LIN {X 0,Y 165.285,Z 372.711,A -85,B 0,C 180,E1 -23309.997,E2 -23309.997} C_VEL
LIN {X 0,Y 164.769,Z 372.772,A -85,B 0,C 180,E1 -23314.891,E2 -23314.891} C_VEL
LIN {X 0,Y 164.844,Z 372.763,A -85,B 0,C 180,E1 -23319.816,E2 -23319.816} C_VEL
LIN {X 0,Y 164.543,Z 372.8,A -85,B 0,C 180,E1 -23324.846,E2 -23324.846} C_VEL
LIN {X 0,Y 164.463,Z 372.807,A -85,B 0,C 180,E1 -23329.987,E2 -23329.987} C_VEL
LIN {X 0,Y 164.382,Z 372.819,A -85,B 0,C 180,E1 -23336.132,E2 -23336.132} C_VEL
LIN {X 0,Y 164.364,Z 372.823,A -85,B 0,C 180,E1 -23341.227,E2 -23341.227} C_VEL
LIN {X 0,Y 164.341,Z 372.821,A -85,B 0,C 180,E1 -23346.773,E2 -23346.773} C_VEL
LIN {X 0,Y 164.367,Z 372.822,A -85,B 0,C 180,E1 -23349.889,E2 -23349.889} C_VEL
LIN {X 0,Y 164.382,Z 372.818,A -85,B 0,C 180,E1 -23353.384,E2 -23353.384} C_VEL
LIN {X 0,Y 164.385,Z 372.819,A -85,B 0,C 180,E1 -23356.843,E2 -23356.843} C_VEL
LIN {X 0,Y 164.365,Z 372.822,A -85,B 0,C 180,E1 -23360.317,E2 -23360.317} C_VEL
LIN {X 0,Y 164.336,Z 372.823,A -85,B 0,C 180,E1 -23364.34,E2 -23364.34} C_VEL
LIN {X 0,Y 164.379,Z 372.819,A -85,B 0,C 180,E1 -23369.135,E2 -23369.135} C_VEL
LIN {X 0,Y 164.413,Z 372.819,A -85,B 0,C 180,E1 -23374.697,E2 -23374.697} C_VEL
LIN {X 0,Y 164.509,Z 372.8,A -85,B 0,C 180,E1 -23380.018,E2 -23380.018} C_VEL
LIN {X 0,Y 164.551,Z 372.798,A -85,B 0,C 180,E1 -23385.154,E2 -23385.154} C_VEL
LIN {X 0,Y 164.842,Z 372.763,A -85,B 0,C 180,E1 -23390.183,E2 -23390.183} C_VEL
LIN {X 0,Y 164.852,Z 372.762,A -85,B 0,C 180,E1 -23392.654,E2 -23392.654} C_VEL
LIN {X 0,Y 165.041,Z 372.736,A -85,B 0,C 180,E1 -23397.562,E2 -23397.562} C_VEL
LIN {X 0,Y 165.286,Z 372.71,A -85,B 0,C 180,E1 -23400.002,E2 -23400.002} C_VEL
LIN {X 0,Y 164.768,Z 372.768,A -85,B 0,C 180,E1 -23404.896,E2 -23404.896} C_VEL
LIN {X 0,Y 164.853,Z 372.762,A -85,B 0,C 180,E1 -23407.35,E2 -23407.35} C_VEL
LIN {X 0,Y 164.742,Z 372.774,A -85,B 0,C 180,E1 -23411.148,E2 -23411.148} C_VEL
LIN {X 0,Y 164.491,Z 372.809,A -85,B 0,C 180,E1 -23417.405,E2 -23417.405} C_VEL
LIN {X 0,Y 164.468,Z 372.806,A -85,B 0,C 180,E1 -23419.992,E2 -23419.992} C_VEL
LIN {X 0,Y 164.388,Z 372.819,A -85,B 0,C 180,E1 -23426.137,E2 -23426.137} C_VEL
LIN {X 0,Y 164.37,Z 372.822,A -85,B 0,C 180,E1 -23431.232,E2 -23431.232} C_VEL
LIN {X 0,Y 164.29,Z 372.83,A -85,B 0,C 180,E1 -23436.793,E2 -23436.793} C_VEL
LIN {X 0,Y 164.289,Z 372.831,A -85,B 0,C 180,E1 -23439.919,E2 -23439.919} C_VEL
LIN {X 0,Y 164.529,Z 372.877,A -85,B 0,C 180,E1 -23446.125,E2 -23446.125} C_VEL
LIN {X 0,Y 165.393,Z 377.162,A -85,B 0,C 180,E1 -23451.969,E2 -23451.969} C_VEL
LIN {X 0,Y 165.659,Z 379.629,A -85,B 0,C 180,E1 -23455.155,E2 -23455.155} C_VEL
LIN {X 0,Y 164.918,Z 382.338,A -85,B 0,C 180,E1 -23458.467,E2 -23458.467} C_VEL
LIN {X 0,Y 163.951,Z 385.365,A -85,B 0,C 180,E1 -23462.135,E2 -23462.135} C_VEL
LIN {X 0,Y 165.313,Z 398.175,A -85,B 0,C 180,E1 -23463.679,E2 -23463.679} C_VEL
LIN {X 0,Y 166.01,Z 408.279,A -85,B 0,C 180,E1 -23465.292,E2 -23465.292} C_VEL
LIN {X 0,Y 166.358,Z 416.947,A -85,B 0,C 180,E1 -23467.001,E2 -23467.001} C_VEL
LIN {X 0,Y 166.469,Z 426.075,A -85,B 0,C 180,E1 -23469.194,E2 -23469.194} C_VEL
LIN {X 0,Y 166.277,Z 432.989,A -85,B 0,C 180,E1 -23471.202,E2 -23471.202} C_VEL
LIN {X 0,Y 164.707,Z 440.811,A -85,B 0,C 180,E1 -23473.901,E2 -23473.901} C_VEL
LIN {X 0,Y 163.462,Z 447.658,A -85,B 0,C 180,E1 -23476.958,E2 -23476.958} C_VEL
LIN {X 0,Y 162.683,Z 453.124,A -85,B 0,C 180,E1 -23480.053,E2 -23480.053} C_VEL
LIN {X 0,Y 162.191,Z 458.179,A -85,B 0,C 180,E1 -23483.784,E2 -23483.784} C_VEL
LIN {X 0,Y 162.156,Z 461.833,A -85,B 0,C 180,E1 -23487.519,E2 -23487.519} C_VEL
LIN {X 0,Y 162.287,Z 463.452,A -85,B 0,C 180,E1 -23490.003,E2 -23490.003} C_VEL
LIN {X 0,Y 161.97,Z 464.904,A -85,B 0,C 180,E1 -23493.61,E2 -23493.61} C_VEL
LIN {X 0,Y 162.138,Z 465.306,A -85,B 0,C 180,E1 -23497.475,E2 -23497.475} C_VEL
LIN {X 0,Y 162.598,Z 464.896,A -85,B 0,C 180,E1 -23499.959,E2 -23499.959} C_VEL
LIN {X 0,Y 163.324,Z 464.018,A -85,B 0,C 180,E1 -23502.428,E2 -23502.428} C_VEL
LIN {X 0,Y 164.353,Z 462.7,A -85,B 0,C 180,E1 -23504.87,E2 -23504.87} C_VEL
LIN {X 0,Y 166.476,Z 459.738,A -85,B 0,C 180,E1 -23508.462,E2 -23508.462} C_VEL
LIN {X 0,Y 169.37,Z 455.573,A -85,B 0,C 180,E1 -23511.932,E2 -23511.932} C_VEL
LIN {X 0,Y 172.955,Z 450.071,A -85,B 0,C 180,E1 -23515.259,E2 -23515.259} C_VEL
LIN {X 0,Y 175.939,Z 444.205,A -85,B 0,C 180,E1 -23517.996,E2 -23517.996} C_VEL
LIN {X 0,Y 178.202,Z 437.103,A -85,B 0,C 180,E1 -23520.847,E2 -23520.847} C_VEL
LIN {X 0,Y 179.47,Z 430.444,A -85,B 0,C 180,E1 -23523.249,E2 -23523.249} C_VEL
LIN {X 0,Y 180.203,Z 422.802,A -85,B 0,C 180,E1 -23525.807,E2 -23525.807} C_VEL
LIN {X 0,Y 180.245,Z 421.902,A -85,B 0,C 180,E1 -23526.094,E2 -23526.094} C_VEL
LIN {X 0,Y 180.072,Z 419.304,A -85,B 0,C 180,E1 -23527.031,E2 -23527.031} C_VEL
LIN {X 0,Y 179.317,Z 417.046,A -85,B 0,C 180,E1 -23528.033,E2 -23528.033} C_VEL
LIN {X 0,Y 176.917,Z 413.276,A -85,B 0,C 180,E1 -23530.156,E2 -23530.156} C_VEL
LIN {X 0,Y 172.898,Z 407.932,A -85,B 0,C 180,E1 -23533.533,E2 -23533.533} C_VEL
LIN {X 0,Y 171.927,Z 405.803,A -85,B 0,C 180,E1 -23534.644,E2 -23534.644} C_VEL
LIN {X 0,Y 169.122,Z 398.872,A -85,B 0,C 180,E1 -23538.422,E2 -23538.422} C_VEL
LIN {X 0,Y 167.171,Z 395.11,A -85,B 0,C 180,E1 -23540.902,E2 -23540.902} C_VEL
LIN {X 0,Y 166.686,Z 393.384,A -85,B 0,C 180,E1 -23541.849,E2 -23541.849} C_VEL
LIN {X 0,Y 164.248,Z 389.736,A -85,B 0,C 180,E1 -23545.195,E2 -23545.195} C_VEL
LIN {X 0,Y 163.031,Z 386.548,A -85,B 0,C 180,E1 -23547.664,E2 -23547.664} C_VEL
LIN {X 0,Y 159.813,Z 382.313,A -85,B 0,C 180,E1 -23555.65,E2 -23555.65} C_VEL
LIN {X 0,Y 159.422,Z 380.964,A -85,B 0,C 180,E1 -23560.691,E2 -23560.691} C_VEL
LIN {X 0,Y 160.286,Z 381.531,A -85,B 0,C 180,E1 -23566.625,E2 -23566.625} C_VEL
LIN {X 0,Y 163.146,Z 383.354,A -85,B 0,C 180,E1 -23572.806,E2 -23572.806} C_VEL
LIN {X 0,Y 164.296,Z 385.761,A -85,B 0,C 180,E1 -23575.09,E2 -23575.09} C_VEL
LIN {X 0,Y 167.058,Z 388.467,A -85,B 0,C 180,E1 -23578.791,E2 -23578.791} C_VEL
LIN {X 0,Y 171.293,Z 396.943,A -85,B 0,C 180,E1 -23584.704,E2 -23584.704} C_VEL
LIN {X 0,Y 173.349,Z 401.847,A -85,B 0,C 180,E1 -23587.539,E2 -23587.539} C_VEL
LIN {X 0,Y 175.255,Z 408.041,A -85,B 0,C 180,E1 -23590.689,E2 -23590.689} C_VEL
LIN {X 0,Y 176.257,Z 414.922,A -85,B 0,C 180,E1 -23593.839,E2 -23593.839} C_VEL
LIN {X 0,Y 176.281,Z 421.806,A -85,B 0,C 180,E1 -23596.888,E2 -23596.888} C_VEL
LIN {X 0,Y 175.611,Z 426.875,A -85,B 0,C 180,E1 -23599.189,E2 -23599.189} C_VEL
LIN {X 0,Y 175.131,Z 428.204,A -85,B 0,C 180,E1 -23599.767,E2 -23599.767} C_VEL
LIN {X 0,Y 171.752,Z 433.94,A -85,B 0,C 180,E1 -23602.123,E2 -23602.123} C_VEL
LIN {X 0,Y 168.512,Z 438.818,A -85,B 0,C 180,E1 -23604.646,E2 -23604.646} C_VEL
LIN {X 0,Y 164.887,Z 443.625,A -85,B 0,C 180,E1 -23607.957,E2 -23607.957} C_VEL
LIN {X 0,Y 161.8,Z 447.187,A -85,B 0,C 180,E1 -23611.412,E2 -23611.412} C_VEL
LIN {X 0,Y 159.242,Z 449.625,A -85,B 0,C 180,E1 -23615.008,E2 -23615.008} C_VEL
LIN {X 0,Y 157.275,Z 450.962,A -85,B 0,C 180,E1 -23618.723,E2 -23618.723} C_VEL
LIN {X 0,Y 155.498,Z 451.005,A -85,B 0,C 180,E1 -23623.681,E2 -23623.681} C_VEL
LIN {X 0,Y 154.826,Z 450.049,A -85,B 0,C 180,E1 -23627.083,E2 -23627.083} C_VEL
LIN {X 0,Y 154.681,Z 447.051,A -85,B 0,C 180,E1 -23632.219,E2 -23632.219} C_VEL
LIN {X 0,Y 155.103,Z 443.465,A -85,B 0,C 180,E1 -23635.93,E2 -23635.93} C_VEL
LIN {X 0,Y 155.766,Z 439.558,A -85,B 0,C 180,E1 -23639.004,E2 -23639.004} C_VEL
LIN {X 0,Y 156.675,Z 434.938,A -85,B 0,C 180,E1 -23641.899,E2 -23641.899} C_VEL
LIN {X 0,Y 157.955,Z 428.745,A -85,B 0,C 180,E1 -23644.992,E2 -23644.992} C_VEL
LIN {X 0,Y 159.061,Z 423.19,A -85,B 0,C 180,E1 -23647.269,E2 -23647.269} C_VEL
LIN {X 0,Y 160.6,Z 415.517,A -85,B 0,C 180,E1 -23649.838,E2 -23649.838} C_VEL
LIN {X 0,Y 162.128,Z 407.481,A -85,B 0,C 180,E1 -23652.006,E2 -23652.006} C_VEL
LIN {X 0,Y 161.25,Z 398.757,A -85,B 0,C 180,E1 -23654.125,E2 -23654.125} C_VEL
LIN {X 0,Y 159.645,Z 387.621,A -85,B 0,C 180,E1 -23656.31,E2 -23656.31} C_VEL
LIN {X 0,Y 157.788,Z 377.801,A -85,B 0,C 180,E1 -23657.853,E2 -23657.853} C_VEL
LIN {X 0,Y 156.746,Z 373.773,A -85,B 0,C 180,E1 -23658.44,E2 -23658.44} C_VEL
LIN {X 0,Y 157.383,Z 373.696,A -85,B 0,C 180,E1 -23662.298,E2 -23662.298} C_VEL
LIN {X 0,Y 157.934,Z 373.626,A -85,B 0,C 180,E1 -23667.446,E2 -23667.446} C_VEL
LIN {X 0,Y 158.246,Z 373.588,A -85,B 0,C 180,E1 -23669.997,E2 -23669.997} C_VEL
LIN {X 0,Y 157.816,Z 373.64,A -85,B 0,C 180,E1 -23677.674,E2 -23677.674} C_VEL
LIN {X 0,Y 157.696,Z 373.65,A -85,B 0,C 180,E1 -23681.359,E2 -23681.359} C_VEL
LIN {X 0,Y 157.468,Z 373.683,A -85,B 0,C 180,E1 -23685.529,E2 -23685.529} C_VEL
LIN {X 0,Y 157.359,Z 373.691,A -85,B 0,C 180,E1 -23690.931,E2 -23690.931} C_VEL
LIN {X 0,Y 157.303,Z 373.7,A -85,B 0,C 180,E1 -23696.683,E2 -23696.683} C_VEL
LIN {X 0,Y 157.266,Z 373.707,A -85,B 0,C 180,E1 -23702.425,E2 -23702.425} C_VEL
LIN {X 0,Y 157.315,Z 373.696,A -85,B 0,C 180,E1 -23706.477,E2 -23706.477} C_VEL
LIN {X 0,Y 157.287,Z 373.703,A -85,B 0,C 180,E1 -23712.081,E2 -23712.081} C_VEL
LIN {X 0,Y 157.302,Z 373.7,A -85,B 0,C 180,E1 -23715.626,E2 -23715.626} C_VEL
LIN {X 0,Y 157.28,Z 373.703,A -85,B 0,C 180,E1 -23721.279,E2 -23721.279} C_VEL
LIN {X 0,Y 157.283,Z 373.702,A -85,B 0,C 180,E1 -23724.49,E2 -23724.49} C_VEL
LIN {X 0,Y 157.282,Z 373.705,A -85,B 0,C 180,E1 -23728.095,E2 -23728.095} C_VEL
LIN {X 0,Y 157.315,Z 373.7,A -85,B 0,C 180,E1 -23733.468,E2 -23733.468} C_VEL
LIN {X 0,Y 157.435,Z 373.68,A -85,B 0,C 180,E1 -23739.617,E2 -23739.617} C_VEL
LIN {X 0,Y 157.479,Z 373.681,A -85,B 0,C 180,E1 -23744.471,E2 -23744.471} C_VEL
LIN {X 0,Y 157.762,Z 373.643,A -85,B 0,C 180,E1 -23749.738,E2 -23749.738} C_VEL
LIN {X 0,Y 157.814,Z 373.64,A -85,B 0,C 180,E1 -23752.325,E2 -23752.325} C_VEL
LIN {X 0,Y 158.248,Z 373.587,A -85,B 0,C 180,E1 -23760.003,E2 -23760.003} C_VEL
LIN {X 0,Y 157.812,Z 373.64,A -85,B 0,C 180,E1 -23767.68,E2 -23767.68} C_VEL
LIN {X 0,Y 157.671,Z 373.656,A -85,B 0,C 180,E1 -23771.317,E2 -23771.317} C_VEL
LIN {X 0,Y 157.456,Z 373.684,A -85,B 0,C 180,E1 -23775.536,E2 -23775.536} C_VEL
LIN {X 0,Y 157.365,Z 373.69,A -85,B 0,C 180,E1 -23780.936,E2 -23780.936} C_VEL
LIN {X 0,Y 157.309,Z 373.701,A -85,B 0,C 180,E1 -23786.688,E2 -23786.688} C_VEL
LIN {X 0,Y 157.27,Z 373.706,A -85,B 0,C 180,E1 -23792.431,E2 -23792.431} C_VEL
LIN {X 0,Y 157.263,Z 373.705,A -85,B 0,C 180,E1 -23796.453,E2 -23796.453} C_VEL
LIN {X 0,Y 157.226,Z 373.712,A -85,B 0,C 180,E1 -23802.109,E2 -23802.109} C_VEL
LIN {X 0,Y 157.506,Z 373.679,A -85,B 0,C 180,E1 -23806.016,E2 -23806.016} C_VEL
LIN {X 0,Y 158.271,Z 377.582,A -85,B 0,C 180,E1 -23811.567,E2 -23811.567} C_VEL
LIN {X 0,Y 158.589,Z 379.982,A -85,B 0,C 180,E1 -23814.827,E2 -23814.827} C_VEL
LIN {X 0,Y 157.992,Z 382.259,A -85,B 0,C 180,E1 -23817.742,E2 -23817.742} C_VEL
LIN {X 0,Y 157.051,Z 385.056,A -85,B 0,C 180,E1 -23821.296,E2 -23821.296} C_VEL
LIN {X 0,Y 158.389,Z 398.191,A -85,B 0,C 180,E1 -23822.981,E2 -23822.981} C_VEL
LIN {X 0,Y 158.988,Z 407.24,A -85,B 0,C 180,E1 -23824.473,E2 -23824.473} C_VEL
LIN {X 0,Y 159.316,Z 416.09,A -85,B 0,C 180,E1 -23826.267,E2 -23826.267} C_VEL
LIN {X 0,Y 159.441,Z 423.58,A -85,B 0,C 180,E1 -23828.097,E2 -23828.097} C_VEL
LIN {X 0,Y 159.372,Z 431.315,A -85,B 0,C 180,E1 -23830.355,E2 -23830.355} C_VEL
LIN {X 0,Y 158.554,Z 436.045,A -85,B 0,C 180,E1 -23831.928,E2 -23831.928} C_VEL
LIN {X 0,Y 157.334,Z 442.433,A -85,B 0,C 180,E1 -23834.457,E2 -23834.457} C_VEL
LIN {X 0,Y 156.328,Z 447.731,A -85,B 0,C 180,E1 -23837.013,E2 -23837.013} C_VEL
LIN {X 0,Y 155.696,Z 452.163,A -85,B 0,C 180,E1 -23839.601,E2 -23839.601} C_VEL
LIN {X 0,Y 155.259,Z 455.836,A -85,B 0,C 180,E1 -23842.199,E2 -23842.199} C_VEL
LIN {X 0,Y 155.08,Z 459.541,A -85,B 0,C 180,E1 -23845.59,E2 -23845.59} C_VEL
LIN {X 0,Y 155.084,Z 461.11,A -85,B 0,C 180,E1 -23847.406,E2 -23847.406} C_VEL
LIN {X 0,Y 155.224,Z 462.836,A -85,B 0,C 180,E1 -23850.003,E2 -23850.003} C_VEL
LIN {X 0,Y 154.902,Z 464.291,A -85,B 0,C 180,E1 -23853.453,E2 -23853.453} C_VEL
LIN {X 0,Y 155.083,Z 464.946,A -85,B 0,C 180,E1 -23857.817,E2 -23857.817} C_VEL
LIN {X 0,Y 155.605,Z 464.613,A -85,B 0,C 180,E1 -23860.412,E2 -23860.412} C_VEL
LIN {X 0,Y 156.381,Z 463.847,A -85,B 0,C 180,E1 -23862.989,E2 -23862.989} C_VEL
LIN {X 0,Y 157.499,Z 462.645,A -85,B 0,C 180,E1 -23865.533,E2 -23865.533} C_VEL
LIN {X 0,Y 159.756,Z 459.824,A -85,B 0,C 180,E1 -23869.268,E2 -23869.268} C_VEL
LIN {X 0,Y 162.809,Z 455.818,A -85,B 0,C 180,E1 -23872.865,E2 -23872.865} C_VEL
LIN {X 0,Y 165.249,Z 452.405,A -85,B 0,C 180,E1 -23875.173,E2 -23875.173} C_VEL
LIN {X 0,Y 168.524,Z 447.242,A -85,B 0,C 180,E1 -23877.947,E2 -23877.947} C_VEL
LIN {X 0,Y 170.516,Z 442.77,A -85,B 0,C 180,E1 -23880.052,E2 -23880.052} C_VEL
LIN {X 0,Y 172.512,Z 436.516,A -85,B 0,C 180,E1 -23882.673,E2 -23882.673} C_VEL
LIN {X 0,Y 173.884,Z 429.558,A -85,B 0,C 180,E1 -23885.331,E2 -23885.331} C_VEL
LIN {X 0,Y 174.626,Z 422.22,A -85,B 0,C 180,E1 -23887.929,E2 -23887.929} C_VEL
LIN {X 0,Y 174.673,Z 415.952,A -85,B 0,C 180,E1 -23890.138,E2 -23890.138} C_VEL
LIN {X 0,Y 173.783,Z 411.346,A -85,B 0,C 180,E1 -23892.037,E2 -23892.037} C_VEL
LIN {X 0,Y 171.927,Z 405.803,A -85,B 0,C 180,E1 -23894.644,E2 -23894.644} C_VEL
LIN {X 0,Y 170.991,Z 403.904,A -85,B 0,C 180,E1 -23895.746,E2 -23895.746} C_VEL
LIN {X 0,Y 169.743,Z 402.527,A -85,B 0,C 180,E1 -23896.911,E2 -23896.911} C_VEL
LIN {X 0,Y 166.812,Z 400.799,A -85,B 0,C 180,E1 -23899.354,E2 -23899.354} C_VEL
LIN {X 0,Y 162.748,Z 398.577,A -85,B 0,C 180,E1 -23903.254,E2 -23903.254} C_VEL
LIN {X 0,Y 161.832,Z 397.323,A -85,B 0,C 180,E1 -23904.566,E2 -23904.566} C_VEL
LIN {X 0,Y 160.311,Z 392.937,A -85,B 0,C 180,E1 -23908.257,E2 -23908.257} C_VEL
LIN {X 0,Y 158.195,Z 390.036,A -85,B 0,C 180,E1 -23913.621,E2 -23913.621} C_VEL
LIN {X 0,Y 157.387,Z 387.899,A -85,B 0,C 180,E1 -23919.683,E2 -23919.683} C_VEL
LIN {X 0,Y 157.738,Z 387.938,A -85,B 0,C 180,E1 -23924.492,E2 -23924.492} C_VEL
LIN {X 0,Y 159.273,Z 389.077,A -85,B 0,C 180,E1 -23929.832,E2 -23929.832} C_VEL
LIN {X 0,Y 160.494,Z 389.995,A -85,B 0,C 180,E1 -23932.449,E2 -23932.449} C_VEL
LIN {X 0,Y 162.076,Z 392.91,A -85,B 0,C 180,E1 -23935.852,E2 -23935.852} C_VEL
LIN {X 0,Y 163.235,Z 394.058,A -85,B 0,C 180,E1 -23937.53,E2 -23937.53} C_VEL
LIN {X 0,Y 164.6,Z 396.861,A -85,B 0,C 180,E1 -23939.998,E2 -23939.998} C_VEL
LIN {X 0,Y 167.475,Z 403.476,A -85,B 0,C 180,E1 -23944.812,E2 -23944.812} C_VEL
LIN {X 0,Y 169.413,Z 409.495,A -85,B 0,C 180,E1 -23948.455,E2 -23948.455} C_VEL
LIN {X 0,Y 170.37,Z 414.917,A -85,B 0,C 180,E1 -23951.297,E2 -23951.297} C_VEL
LIN {X 0,Y 170.554,Z 420.996,A -85,B 0,C 180,E1 -23954.312,E2 -23954.312} C_VEL
LIN {X 0,Y 170.038,Z 426.114,A -85,B 0,C 180,E1 -23956.815,E2 -23956.815} C_VEL
LIN {X 0,Y 169.16,Z 429.719,A -85,B 0,C 180,E1 -23958.591,E2 -23958.591} C_VEL
LIN {X 0,Y 165.611,Z 435.223,A -85,B 0,C 180,E1 -23960.988,E2 -23960.988} C_VEL
LIN {X 0,Y 161.643,Z 440.657,A -85,B 0,C 180,E1 -23964.063,E2 -23964.063} C_VEL
LIN {X 0,Y 158.138,Z 444.855,A -85,B 0,C 180,E1 -23967.266,E2 -23967.266} C_VEL
LIN {X 0,Y 155.123,Z 447.974,A -85,B 0,C 180,E1 -23970.586,E2 -23970.586} C_VEL
LIN {X 0,Y 152.617,Z 450.094,A -85,B 0,C 180,E1 -23974.009,E2 -23974.009} C_VEL
LIN {X 0,Y 150.657,Z 451.288,A -85,B 0,C 180,E1 -23977.525,E2 -23977.525} C_VEL
LIN {X 0,Y 149.076,Z 451.591,A -85,B 0,C 180,E1 -23981.297,E2 -23981.297} C_VEL
LIN {X 0,Y 147.984,Z 450.79,A -85,B 0,C 180,E1 -23985.424,E2 -23985.424} C_VEL
LIN {X 0,Y 147.529,Z 448.816,A -85,B 0,C 180,E1 -23989.655,E2 -23989.655} C_VEL
LIN {X 0,Y 147.569,Z 447.478,A -85,B 0,C 180,E1 -23991.744,E2 -23991.744} C_VEL
LIN {X 0,Y 147.884,Z 444.385,A -85,B 0,C 180,E1 -23995.226,E2 -23995.226} C_VEL
LIN {X 0,Y 148.78,Z 439.15,A -85,B 0,C 180,E1 -23999.479,E2 -23999.479} C_VEL
LIN {X 0,Y 149.55,Z 435.318,A -85,B 0,C 180,E1 -24001.966,E2 -24001.966} C_VEL
LIN {X 0,Y 150.855,Z 429.126,A -85,B 0,C 180,E1 -24005.207,E2 -24005.207} C_VEL
LIN {X 0,Y 152.018,Z 423.532,A -85,B 0,C 180,E1 -24007.604,E2 -24007.604} C_VEL
LIN {X 0,Y 153.327,Z 417.122,A -85,B 0,C 180,E1 -24009.89,E2 -24009.89} C_VEL
LIN {X 0,Y 154.956,Z 408.973,A -85,B 0,C 180,E1 -24012.25,E2 -24012.25} C_VEL
LIN {X 0,Y 155.068,Z 406.477,A -85,B 0,C 180,E1 -24012.935,E2 -24012.935} C_VEL
LIN {X 0,Y 153.893,Z 396.06,A -85,B 0,C 180,E1 -24015.45,E2 -24015.45} C_VEL
LIN {X 0,Y 152.541,Z 387.141,A -85,B 0,C 180,E1 -24017.219,E2 -24017.219} C_VEL
LIN {X 0,Y 150.857,Z 378.629,A -85,B 0,C 180,E1 -24018.646,E2 -24018.646} C_VEL
LIN {X 0,Y 149.857,Z 374.63,A -85,B 0,C 180,E1 -24019.32,E2 -24019.32} C_VEL
LIN {X 0,Y 150.268,Z 374.581,A -85,B 0,C 180,E1 -24021.931,E2 -24021.931} C_VEL
LIN {X 0,Y 150.849,Z 374.509,A -85,B 0,C 180,E1 -24027.326,E2 -24027.326} C_VEL
LIN {X 0,Y 151.205,Z 374.465,A -85,B 0,C 180,E1 -24029.997,E2 -24029.997} C_VEL
LIN {X 0,Y 150.754,Z 374.519,A -85,B 0,C 180,E1 -24038.036,E2 -24038.036} C_VEL
LIN {X 0,Y 150.625,Z 374.53,A -85,B 0,C 180,E1 -24041.542,E2 -24041.542} C_VEL
LIN {X 0,Y 150.373,Z 374.566,A -85,B 0,C 180,E1 -24046.282,E2 -24046.282} C_VEL
LIN {X 0,Y 150.34,Z 374.565,A -85,B 0,C 180,E1 -24050.79,E2 -24050.79} C_VEL
LIN {X 0,Y 150.233,Z 374.58,A -85,B 0,C 180,E1 -24057.28,E2 -24057.28} C_VEL
LIN {X 0,Y 150.207,Z 374.586,A -85,B 0,C 180,E1 -24062.633,E2 -24062.633} C_VEL
LIN {X 0,Y 150.227,Z 374.581,A -85,B 0,C 180,E1 -24067.453,E2 -24067.453} C_VEL
LIN {X 0,Y 150.228,Z 374.584,A -85,B 0,C 180,E1 -24071.543,E2 -24071.543} C_VEL
LIN {X 0,Y 150.278,Z 374.575,A -85,B 0,C 180,E1 -24075.457,E2 -24075.457} C_VEL
LIN {X 0,Y 150.226,Z 374.585,A -85,B 0,C 180,E1 -24079.088,E2 -24079.088} C_VEL
LIN {X 0,Y 150.228,Z 374.58,A -85,B 0,C 180,E1 -24082.677,E2 -24082.677} C_VEL
LIN {X 0,Y 150.207,Z 374.586,A -85,B 0,C 180,E1 -24087.366,E2 -24087.366} C_VEL
LIN {X 0,Y 150.235,Z 374.581,A -85,B 0,C 180,E1 -24092.717,E2 -24092.717} C_VEL
LIN {X 0,Y 150.379,Z 374.559,A -85,B 0,C 180,E1 -24099.169,E2 -24099.169} C_VEL
LIN {X 0,Y 150.388,Z 374.564,A -85,B 0,C 180,E1 -24103.719,E2 -24103.719} C_VEL
LIN {X 0,Y 150.678,Z 374.525,A -85,B 0,C 180,E1 -24109.25,E2 -24109.25} C_VEL
LIN {X 0,Y 150.752,Z 374.52,A -85,B 0,C 180,E1 -24111.963,E2 -24111.963} C_VEL
LIN {X 0,Y 151.209,Z 374.464,A -85,B 0,C 180,E1 -24120.003,E2 -24120.003} C_VEL
LIN {X 0,Y 150.748,Z 374.52,A -85,B 0,C 180,E1 -24128.042,E2 -24128.042} C_VEL
LIN {X 0,Y 150.606,Z 374.534,A -85,B 0,C 180,E1 -24131.51,E2 -24131.51} C_VEL
LIN {X 0,Y 150.364,Z 374.567,A -85,B 0,C 180,E1 -24136.289,E2 -24136.289} C_VEL
LIN {X 0,Y 150.346,Z 374.564,A -85,B 0,C 180,E1 -24140.797,E2 -24140.797} C_VEL
LIN {X 0,Y 150.239,Z 374.581,A -85,B 0,C 180,E1 -24147.286,E2 -24147.286} C_VEL
LIN {X 0,Y 150.21,Z 374.586,A -85,B 0,C 180,E1 -24152.636,E2 -24152.636} C_VEL
LIN {X 0,Y 150.169,Z 374.587,A -85,B 0,C 180,E1 -24157.477,E2 -24157.477} C_VEL
LIN {X 0,Y 150.161,Z 374.592,A -85,B 0,C 180,E1 -24161.515,E2 -24161.515} C_VEL
LIN {X 0,Y 150.488,Z 374.661,A -85,B 0,C 180,E1 -24166.187,E2 -24166.187} C_VEL
LIN {X 0,Y 151.26,Z 378.692,A -85,B 0,C 180,E1 -24172.177,E2 -24172.177} C_VEL
LIN {X 0,Y 151.48,Z 380.375,A -85,B 0,C 180,E1 -24174.558,E2 -24174.558} C_VEL
LIN {X 0,Y 151.124,Z 382.059,A -85,B 0,C 180,E1 -24176.837,E2 -24176.837} C_VEL
LIN {X 0,Y 150.118,Z 384.782,A -85,B 0,C 180,E1 -24180.465,E2 -24180.465} C_VEL
LIN {X 0,Y 151.402,Z 397.721,A -85,B 0,C 180,E1 -24182.159,E2 -24182.159} C_VEL
LIN {X 0,Y 151.982,Z 406.007,A -85,B 0,C 180,E1 -24183.575,E2 -24183.575} C_VEL
LIN {X 0,Y 152.322,Z 415.052,A -85,B 0,C 180,E1 -24185.469,E2 -24185.469} C_VEL
LIN {X 0,Y 152.438,Z 423.314,A -85,B 0,C 180,E1 -24187.569,E2 -24187.569} C_VEL
LIN {X 0,Y 152.347,Z 430.539,A -85,B 0,C 180,E1 -24189.762,E2 -24189.762} C_VEL
LIN {X 0,Y 151.83,Z 434.523,A -85,B 0,C 180,E1 -24191.098,E2 -24191.098} C_VEL
LIN {X 0,Y 150.465,Z 441.089,A -85,B 0,C 180,E1 -24193.729,E2 -24193.729} C_VEL
LIN {X 0,Y 149.216,Z 447.73,A -85,B 0,C 180,E1 -24197.076,E2 -24197.076} C_VEL
LIN {X 0,Y 148.449,Z 453.044,A -85,B 0,C 180,E1 -24200.466,E2 -24200.466} C_VEL
LIN {X 0,Y 148.079,Z 456.458,A -85,B 0,C 180,E1 -24203.189,E2 -24203.189} C_VEL
LIN {X 0,Y 148.027,Z 458.989,A -85,B 0,C 180,E1 -24205.612,E2 -24205.612} C_VEL
LIN {X 0,Y 148.16,Z 462.213,A -85,B 0,C 180,E1 -24210.003,E2 -24210.003} C_VEL
LIN {X 0,Y 147.844,Z 463.697,A -85,B 0,C 180,E1 -24213.341,E2 -24213.341} C_VEL
LIN {X 0,Y 147.843,Z 464.321,A -85,B 0,C 180,E1 -24215.459,E2 -24215.459} C_VEL
LIN {X 0,Y 148.037,Z 464.549,A -85,B 0,C 180,E1 -24218.192,E2 -24218.192} C_VEL
LIN {X 0,Y 148.608,Z 464.331,A -85,B 0,C 180,E1 -24220.908,E2 -24220.908} C_VEL
LIN {X 0,Y 149.465,Z 463.69,A -85,B 0,C 180,E1 -24223.601,E2 -24223.601} C_VEL
LIN {X 0,Y 150.652,Z 462.6,A -85,B 0,C 180,E1 -24226.258,E2 -24226.258} C_VEL
LIN {X 0,Y 153.075,Z 459.93,A -85,B 0,C 180,E1 -24230.145,E2 -24230.145} C_VEL
LIN {X 0,Y 156.3,Z 456.061,A -85,B 0,C 180,E1 -24233.875,E2 -24233.875} C_VEL
LIN {X 0,Y 160.27,Z 450.887,A -85,B 0,C 180,E1 -24237.419,E2 -24237.419} C_VEL
LIN {X 0,Y 162.821,Z 446.85,A -85,B 0,C 180,E1 -24239.624,E2 -24239.624} C_VEL
LIN {X 0,Y 165.124,Z 441.709,A -85,B 0,C 180,E1 -24242.144,E2 -24242.144} C_VEL
LIN {X 0,Y 166.951,Z 436.041,A -85,B 0,C 180,E1 -24244.635,E2 -24244.635} C_VEL
LIN {X 0,Y 168.436,Z 428.775,A -85,B 0,C 180,E1 -24247.552,E2 -24247.552} C_VEL
LIN {X 0,Y 169.213,Z 422.018,A -85,B 0,C 180,E1 -24250.142,E2 -24250.142} C_VEL
LIN {X 0,Y 169.101,Z 417.161,A -85,B 0,C 180,E1 -24252.149,E2 -24252.149} C_VEL
LIN {X 0,Y 167.294,Z 410.422,A -85,B 0,C 180,E1 -24255.579,E2 -24255.579} C_VEL
LIN {X 0,Y 164.999,Z 404.173,A -85,B 0,C 180,E1 -24259.271,E2 -24259.271} C_VEL
LIN {X 0,Y 163.008,Z 399.017,A -85,B 0,C 180,E1 -24262.869,E2 -24262.869} C_VEL
LIN {X 0,Y 161.832,Z 397.323,A -85,B 0,C 180,E1 -24264.566,E2 -24264.566} C_VEL
LIN {X 0,Y 160.543,Z 395.876,A -85,B 0,C 180,E1 -24266.545,E2 -24266.545} C_VEL
LIN {X 0,Y 158.987,Z 395.532,A -85,B 0,C 180,E1 -24268.6,E2 -24268.6} C_VEL
LIN {X 0,Y 155.455,Z 396.122,A -85,B 0,C 180,E1 -24274.329,E2 -24274.329} C_VEL
LIN {X 0,Y 155.077,Z 395.767,A -85,B 0,C 180,E1 -24275.803,E2 -24275.803} C_VEL
LIN {X 0,Y 154.837,Z 394.827,A -85,B 0,C 180,E1 -24278.706,E2 -24278.706} C_VEL
LIN {X 0,Y 154.892,Z 394.404,A -85,B 0,C 180,E1 -24282.344,E2 -24282.344} C_VEL
LIN {X 0,Y 155.624,Z 394.948,A -85,B 0,C 180,E1 -24286.948,E2 -24286.948} C_VEL
LIN {X 0,Y 156.81,Z 395.842,A -85,B 0,C 180,E1 -24290.421,E2 -24290.421} C_VEL
LIN {X 0,Y 157.539,Z 396.61,A -85,B 0,C 180,E1 -24292.306,E2 -24292.306} C_VEL
LIN {X 0,Y 158.417,Z 398.721,A -85,B 0,C 180,E1 -24294.907,E2 -24294.907} C_VEL
LIN {X 0,Y 159.844,Z 400.412,A -85,B 0,C 180,E1 -24297.478,E2 -24297.478} C_VEL
LIN {X 0,Y 161.535,Z 404.863,A -85,B 0,C 180,E1 -24301.318,E2 -24301.318} C_VEL
LIN {X 0,Y 163.268,Z 409.677,A -85,B 0,C 180,E1 -24304.936,E2 -24304.936} C_VEL
LIN {X 0,Y 164.523,Z 415.377,A -85,B 0,C 180,E1 -24308.596,E2 -24308.596} C_VEL
LIN {X 0,Y 164.85,Z 420.122,A -85,B 0,C 180,E1 -24311.304,E2 -24311.304} C_VEL
LIN {X 0,Y 164.519,Z 425.494,A -85,B 0,C 180,E1 -24314.216,E2 -24314.216} C_VEL
LIN {X 0,Y 163.489,Z 430.396,A -85,B 0,C 180,E1 -24316.865,E2 -24316.865} C_VEL
LIN {X 0,Y 162.433,Z 432.501,A -85,B 0,C 180,E1 -24317.839,E2 -24317.839} C_VEL
LIN {X 0,Y 158.002,Z 438.654,A -85,B 0,C 180,E1 -24320.911,E2 -24320.911} C_VEL
LIN {X 0,Y 153.76,Z 443.57,A -85,B 0,C 180,E1 -24324.288,E2 -24324.288} C_VEL
LIN {X 0,Y 150.015,Z 447.322,A -85,B 0,C 180,E1 -24327.933,E2 -24327.933} C_VEL
LIN {X 0,Y 147.49,Z 449.466,A -85,B 0,C 180,E1 -24330.933,E2 -24330.933} C_VEL
LIN {X 0,Y 144.344,Z 451.469,A -85,B 0,C 180,E1 -24335.748,E2 -24335.748} C_VEL
LIN {X 0,Y 142.443,Z 451.96,A -85,B 0,C 180,E1 -24339.893,E2 -24339.893} C_VEL
LIN {X 0,Y 141.133,Z 451.306,A -85,B 0,C 180,E1 -24344.195,E2 -24344.195} C_VEL
LIN {X 0,Y 140.441,Z 448.97,A -85,B 0,C 180,E1 -24349.412,E2 -24349.412} C_VEL
LIN {X 0,Y 140.558,Z 446.312,A -85,B 0,C 180,E1 -24353.125,E2 -24353.125} C_VEL
LIN {X 0,Y 141.017,Z 442.783,A -85,B 0,C 180,E1 -24356.751,E2 -24356.751} C_VEL
LIN {X 0,Y 141.872,Z 438.302,A -85,B 0,C 180,E1 -24360.301,E2 -24360.301} C_VEL
LIN {X 0,Y 143.37,Z 431.237,A -85,B 0,C 180,E1 -24364.597,E2 -24364.597} C_VEL
LIN {X 0,Y 145.025,Z 423.68,A -85,B 0,C 180,E1 -24368.049,E2 -24368.049} C_VEL
LIN {X 0,Y 146.313,Z 417.512,A -85,B 0,C 180,E1 -24370.349,E2 -24370.349} C_VEL
LIN {X 0,Y 148.053,Z 409.218,A -85,B 0,C 180,E1 -24372.855,E2 -24372.855} C_VEL
LIN {X 0,Y 147.82,Z 404.136,A -85,B 0,C 180,E1 -24374.282,E2 -24374.282} C_VEL
LIN {X 0,Y 146.719,Z 394.89,A -85,B 0,C 180,E1 -24376.528,E2 -24376.528} C_VEL
LIN {X 0,Y 145.448,Z 386.406,A -85,B 0,C 180,E1 -24378.243,E2 -24378.243} C_VEL
LIN {X 0,Y 143.749,Z 378.858,A -85,B 0,C 180,E1 -24379.582,E2 -24379.582} C_VEL
LIN {X 0,Y 142.942,Z 375.493,A -85,B 0,C 180,E1 -24380.196,E2 -24380.196} C_VEL
LIN {X 0,Y 143.415,Z 375.437,A -85,B 0,C 180,E1 -24384.372,E2 -24384.372} C_VEL
LIN {X 0,Y 144.162,Z 375.343,A -85,B 0,C 180,E1 -24389.996,E2 -24389.996} C_VEL
LIN {X 0,Y 143.676,Z 375.4,A -85,B 0,C 180,E1 -24398.435,E2 -24398.435} C_VEL
LIN {X 0,Y 143.562,Z 375.41,A -85,B 0,C 180,E1 -24401.755,E2 -24401.755} C_VEL
LIN {X 0,Y 143.306,Z 375.446,A -85,B 0,C 180,E1 -24407.109,E2 -24407.109} C_VEL
LIN {X 0,Y 143.266,Z 375.447,A -85,B 0,C 180,E1 -24411.252,E2 -24411.252} C_VEL
LIN {X 0,Y 143.179,Z 375.456,A -85,B 0,C 180,E1 -24417.935,E2 -24417.935} C_VEL
LIN {X 0,Y 143.159,Z 375.465,A -85,B 0,C 180,E1 -24423.435,E2 -24423.435} C_VEL
LIN {X 0,Y 143.121,Z 375.469,A -85,B 0,C 180,E1 -24429.665,E2 -24429.665} C_VEL
LIN {X 0,Y 143.172,Z 375.459,A -85,B 0,C 180,E1 -24433.406,E2 -24433.406} C_VEL
LIN {X 0,Y 143.159,Z 375.465,A -85,B 0,C 180,E1 -24437.418,E2 -24437.418} C_VEL
LIN {X 0,Y 143.157,Z 375.461,A -85,B 0,C 180,E1 -24441.759,E2 -24441.759} C_VEL
LIN {X 0,Y 143.174,Z 375.463,A -85,B 0,C 180,E1 -24447.323,E2 -24447.323} C_VEL
LIN {X 0,Y 143.154,Z 375.464,A -85,B 0,C 180,E1 -24453.782,E2 -24453.782} C_VEL
LIN {X 0,Y 143.333,Z 375.437,A -85,B 0,C 180,E1 -24459.929,E2 -24459.929} C_VEL
LIN {X 0,Y 143.377,Z 375.437,A -85,B 0,C 180,E1 -24465.816,E2 -24465.816} C_VEL
LIN {X 0,Y 143.592,Z 375.408,A -85,B 0,C 180,E1 -24468.713,E2 -24468.713} C_VEL
LIN {X 0,Y 143.674,Z 375.4,A -85,B 0,C 180,E1 -24471.564,E2 -24471.564} C_VEL
LIN {X 0,Y 144.168,Z 375.341,A -85,B 0,C 180,E1 -24480.003,E2 -24480.003} C_VEL
LIN {X 0,Y 143.667,Z 375.401,A -85,B 0,C 180,E1 -24488.442,E2 -24488.442} C_VEL
LIN {X 0,Y 143.54,Z 375.413,A -85,B 0,C 180,E1 -24491.716,E2 -24491.716} C_VEL
LIN {X 0,Y 143.302,Z 375.447,A -85,B 0,C 180,E1 -24497.116,E2 -24497.116} C_VEL
LIN {X 0,Y 143.271,Z 375.446,A -85,B 0,C 180,E1 -24501.259,E2 -24501.259} C_VEL
LIN {X 0,Y 143.185,Z 375.457,A -85,B 0,C 180,E1 -24507.941,E2 -24507.941} C_VEL
LIN {X 0,Y 143.16,Z 375.465,A -85,B 0,C 180,E1 -24513.437,E2 -24513.437} C_VEL
LIN {X 0,Y 143.063,Z 375.475,A -85,B 0,C 180,E1 -24519.693,E2 -24519.693} C_VEL
LIN {X 0,Y 143.436,Z 375.498,A -85,B 0,C 180,E1 -24526.184,E2 -24526.184} C_VEL
LIN {X 0,Y 144.056,Z 378.782,A -85,B 0,C 180,E1 -24531.317,E2 -24531.317} C_VEL
LIN {X 0,Y 144.374,Z 380.752,A -85,B 0,C 180,E1 -24534.262,E2 -24534.262} C_VEL
LIN {X 0,Y 144.253,Z 381.905,A -85,B 0,C 180,E1 -24535.922,E2 -24535.922} C_VEL
LIN {X 0,Y 143.228,Z 384.46,A -85,B 0,C 180,E1 -24539.504,E2 -24539.504} C_VEL
LIN {X 0,Y 144.42,Z 396.684,A -85,B 0,C 180,E1 -24541.161,E2 -24541.161} C_VEL
LIN {X 0,Y 145.058,Z 405.901,A -85,B 0,C 180,E1 -24542.824,E2 -24542.824} C_VEL
LIN {X 0,Y 145.361,Z 415.59,A -85,B 0,C 180,E1 -24544.982,E2 -24544.982} C_VEL
LIN {X 0,Y 145.414,Z 423.959,A -85,B 0,C 180,E1 -24547.258,E2 -24547.258} C_VEL
LIN {X 0,Y 145.272,Z 431.84,A -85,B 0,C 180,E1 -24549.841,E2 -24549.841} C_VEL
LIN {X 0,Y 143.641,Z 439.698,A -85,B 0,C 180,E1 -24552.932,E2 -24552.932} C_VEL
LIN {X 0,Y 142.281,Z 446.559,A -85,B 0,C 180,E1 -24556.434,E2 -24556.434} C_VEL
LIN {X 0,Y 141.451,Z 452.028,A -85,B 0,C 180,E1 -24559.989,E2 -24559.989} C_VEL
LIN {X 0,Y 140.935,Z 457.078,A -85,B 0,C 180,E1 -24564.28,E2 -24564.28} C_VEL
LIN {X 0,Y 140.937,Z 459.619,A -85,B 0,C 180,E1 -24567.145,E2 -24567.145} C_VEL
LIN {X 0,Y 141.096,Z 461.586,A -85,B 0,C 180,E1 -24570.004,E2 -24570.004} C_VEL
LIN {X 0,Y 140.779,Z 463.076,A -85,B 0,C 180,E1 -24573.156,E2 -24573.156} C_VEL
LIN {X 0,Y 140.78,Z 463.819,A -85,B 0,C 180,E1 -24575.734,E2 -24575.734} C_VEL
LIN {X 0,Y 141.012,Z 464.147,A -85,B 0,C 180,E1 -24578.603,E2 -24578.603} C_VEL
LIN {X 0,Y 141.636,Z 464.054,A -85,B 0,C 180,E1 -24581.452,E2 -24581.452} C_VEL
LIN {X 0,Y 142.557,Z 463.537,A -85,B 0,C 180,E1 -24584.274,E2 -24584.274} C_VEL
LIN {X 0,Y 143.839,Z 462.479,A -85,B 0,C 180,E1 -24587.051,E2 -24587.051} C_VEL
LIN {X 0,Y 146.41,Z 460.021,A -85,B 0,C 180,E1 -24591.105,E2 -24591.105} C_VEL
LIN {X 0,Y 149.845,Z 456.34,A -85,B 0,C 180,E1 -24594.972,E2 -24594.972} C_VEL
LIN {X 0,Y 152.57,Z 453.242,A -85,B 0,C 180,E1 -24597.432,E2 -24597.432} C_VEL
LIN {X 0,Y 156.182,Z 448.411,A -85,B 0,C 180,E1 -24600.417,E2 -24600.417} C_VEL
LIN {X 0,Y 159.126,Z 442.561,A -85,B 0,C 180,E1 -24603.512,E2 -24603.512} C_VEL
LIN {X 0,Y 161.111,Z 437.152,A -85,B 0,C 180,E1 -24606.082,E2 -24606.082} C_VEL
LIN {X 0,Y 163.085,Z 428.986,A -85,B 0,C 180,E1 -24609.604,E2 -24609.604} C_VEL
LIN {X 0,Y 163.818,Z 423.238,A -85,B 0,C 180,E1 -24612.034,E2 -24612.034} C_VEL
LIN {X 0,Y 163.59,Z 420.324,A -85,B 0,C 180,E1 -24613.427,E2 -24613.427} C_VEL
LIN {X 0,Y 162.209,Z 414.194,A -85,B 0,C 180,E1 -24616.966,E2 -24616.966} C_VEL
LIN {X 0,Y 160.613,Z 409.085,A -85,B 0,C 180,E1 -24620.383,E2 -24620.383} C_VEL
LIN {X 0,Y 159.276,Z 404.852,A -85,B 0,C 180,E1 -24623.434,E2 -24623.434} C_VEL
LIN {X 0,Y 157.921,Z 402.181,A -85,B 0,C 180,E1 -24626.176,E2 -24626.176} C_VEL
LIN {X 0,Y 157.431,Z 400.067,A -85,B 0,C 180,E1 -24628.021,E2 -24628.021} C_VEL
LIN {X 0,Y 156.529,Z 398.372,A -85,B 0,C 180,E1 -24630.401,E2 -24630.401} C_VEL
LIN {X 0,Y 155.077,Z 395.767,A -85,B 0,C 180,E1 -24635.803,E2 -24635.803} C_VEL
LIN {X 0,Y 154.621,Z 395.661,A -85,B 0,C 180,E1 -24637.976,E2 -24637.976} C_VEL
LIN {X 0,Y 153.941,Z 396.672,A -85,B 0,C 180,E1 -24640.137,E2 -24640.137} C_VEL
LIN {X 0,Y 152.462,Z 400.877,A -85,B 0,C 180,E1 -24645.928,E2 -24645.928} C_VEL
LIN {X 0,Y 152.639,Z 401.441,A -85,B 0,C 180,E1 -24647.422,E2 -24647.422} C_VEL
LIN {X 0,Y 153.256,Z 401.886,A -85,B 0,C 180,E1 -24649.428,E2 -24649.428} C_VEL
LIN {X 0,Y 154.154,Z 402.96,A -85,B 0,C 180,E1 -24652.136,E2 -24652.136} C_VEL
LIN {X 0,Y 156.067,Z 406.563,A -85,B 0,C 180,E1 -24657.416,E2 -24657.416} C_VEL
LIN {X 0,Y 157.516,Z 411.51,A -85,B 0,C 180,E1 -24661.865,E2 -24661.865} C_VEL
LIN {X 0,Y 158.573,Z 415.549,A -85,B 0,C 180,E1 -24665.083,E2 -24665.083} C_VEL
LIN {X 0,Y 159.231,Z 421.072,A -85,B 0,C 180,E1 -24668.884,E2 -24668.884} C_VEL
LIN {X 0,Y 158.969,Z 425.721,A -85,B 0,C 180,E1 -24671.728,E2 -24671.728} C_VEL
LIN {X 0,Y 158.265,Z 429.8,A -85,B 0,C 180,E1 -24674.133,E2 -24674.133} C_VEL
LIN {X 0,Y 157.586,Z 432.109,A -85,B 0,C 180,E1 -24675.518,E2 -24675.518} C_VEL
LIN {X 0,Y 156.551,Z 434.074,A -85,B 0,C 180,E1 -24676.511,E2 -24676.511} C_VEL
LIN {X 0,Y 151.763,Z 439.998,A -85,B 0,C 180,E1 -24679.756,E2 -24679.756} C_VEL
LIN {X 0,Y 148.491,Z 443.558,A -85,B 0,C 180,E1 -24682.246,E2 -24682.246} C_VEL
LIN {X 0,Y 144.4,Z 447.407,A -85,B 0,C 180,E1 -24685.975,E2 -24685.975} C_VEL
LIN {X 0,Y 140.889,Z 450.109,A -85,B 0,C 180,E1 -24689.919,E2 -24689.919} C_VEL
LIN {X 0,Y 138.053,Z 451.725,A -85,B 0,C 180,E1 -24694.051,E2 -24694.051} C_VEL
LIN {X 0,Y 135.618,Z 452.319,A -85,B 0,C 180,E1 -24698.978,E2 -24698.978} C_VEL
LIN {X 0,Y 134.33,Z 451.775,A -85,B 0,C 180,E1 -24702.902,E2 -24702.902} C_VEL
LIN {X 0,Y 133.478,Z 450.053,A -85,B 0,C 180,E1 -24707.483,E2 -24707.483} C_VEL
LIN {X 0,Y 133.382,Z 447.043,A -85,B 0,C 180,E1 -24712.214,E2 -24712.214} C_VEL
LIN {X 0,Y 133.774,Z 443.704,A -85,B 0,C 180,E1 -24715.963,E2 -24715.963} C_VEL
LIN {X 0,Y 134.736,Z 438.605,A -85,B 0,C 180,E1 -24720.293,E2 -24720.293} C_VEL
LIN {X 0,Y 136.289,Z 431.504,A -85,B 0,C 180,E1 -24724.818,E2 -24724.818} C_VEL
LIN {X 0,Y 137.996,Z 423.967,A -85,B 0,C 180,E1 -24728.433,E2 -24728.433} C_VEL
LIN {X 0,Y 139.552,Z 416.782,A -85,B 0,C 180,E1 -24731.2,E2 -24731.2} C_VEL
LIN {X 0,Y 141.064,Z 409.937,A -85,B 0,C 180,E1 -24733.349,E2 -24733.349} C_VEL
LIN {X 0,Y 140.88,Z 405.039,A -85,B 0,C 180,E1 -24734.813,E2 -24734.813} C_VEL
LIN {X 0,Y 139.868,Z 396.049,A -85,B 0,C 180,E1 -24737.131,E2 -24737.131} C_VEL
LIN {X 0,Y 138.542,Z 386.997,A -85,B 0,C 180,E1 -24739.086,E2 -24739.086} C_VEL
LIN {X 0,Y 136.559,Z 378.646,A -85,B 0,C 180,E1 -24740.673,E2 -24740.673} C_VEL
LIN {X 0,Y 136.018,Z 376.356,A -85,B 0,C 180,E1 -24741.079,E2 -24741.079} C_VEL
LIN {X 0,Y 136.673,Z 376.275,A -85,B 0,C 180,E1 -24747.049,E2 -24747.049} C_VEL
LIN {X 0,Y 137.116,Z 376.22,A -85,B 0,C 180,E1 -24749.996,E2 -24749.996} C_VEL
LIN {X 0,Y 136.6,Z 376.281,A -85,B 0,C 180,E1 -24758.875,E2 -24758.875} C_VEL
LIN {X 0,Y 136.483,Z 376.291,A -85,B 0,C 180,E1 -24761.954,E2 -24761.954} C_VEL
LIN {X 0,Y 136.242,Z 376.324,A -85,B 0,C 180,E1 -24768.025,E2 -24768.025} C_VEL
LIN {X 0,Y 136.187,Z 376.331,A -85,B 0,C 180,E1 -24771.746,E2 -24771.746} C_VEL
LIN {X 0,Y 136.089,Z 376.339,A -85,B 0,C 180,E1 -24778.614,E2 -24778.614} C_VEL
LIN {X 0,Y 136.072,Z 376.346,A -85,B 0,C 180,E1 -24784.616,E2 -24784.616} C_VEL
LIN {X 0,Y 136.095,Z 376.345,A -85,B 0,C 180,E1 -24789.236,E2 -24789.236} C_VEL
LIN {X 0,Y 136.107,Z 376.338,A -85,B 0,C 180,E1 -24793.71,E2 -24793.71} C_VEL
LIN {X 0,Y 136.106,Z 376.343,A -85,B 0,C 180,E1 -24797.839,E2 -24797.839} C_VEL
LIN {X 0,Y 136.108,Z 376.339,A -85,B 0,C 180,E1 -24801.715,E2 -24801.715} C_VEL
LIN {X 0,Y 136.081,Z 376.345,A -85,B 0,C 180,E1 -24805.716,E2 -24805.716} C_VEL
LIN {X 0,Y 136.137,Z 376.335,A -85,B 0,C 180,E1 -24812.318,E2 -24812.318} C_VEL
LIN {X 0,Y 136.267,Z 376.317,A -85,B 0,C 180,E1 -24818.84,E2 -24818.84} C_VEL
LIN {X 0,Y 136.284,Z 376.32,A -85,B 0,C 180,E1 -24825.061,E2 -24825.061} C_VEL
LIN {X 0,Y 136.491,Z 376.29,A -85,B 0,C 180,E1 -24828.117,E2 -24828.117} C_VEL
LIN {X 0,Y 136.598,Z 376.281,A -85,B 0,C 180,E1 -24831.124,E2 -24831.124} C_VEL
LIN {X 0,Y 137.125,Z 376.218,A -85,B 0,C 180,E1 -24840.003,E2 -24840.003} C_VEL
LIN {X 0,Y 136.591,Z 376.282,A -85,B 0,C 180,E1 -24848.882,E2 -24848.882} C_VEL
LIN {X 0,Y 136.483,Z 376.29,A -85,B 0,C 180,E1 -24851.958,E2 -24851.958} C_VEL
LIN {X 0,Y 136.24,Z 376.325,A -85,B 0,C 180,E1 -24858.033,E2 -24858.033} C_VEL
LIN {X 0,Y 136.193,Z 376.329,A -85,B 0,C 180,E1 -24861.754,E2 -24861.754} C_VEL
LIN {X 0,Y 136.095,Z 376.34,A -85,B 0,C 180,E1 -24868.621,E2 -24868.621} C_VEL
LIN {X 0,Y 136.066,Z 376.348,A -85,B 0,C 180,E1 -24874.625,E2 -24874.625} C_VEL
LIN {X 0,Y 136.032,Z 376.351,A -85,B 0,C 180,E1 -24879.205,E2 -24879.205} C_VEL
LIN {X 0,Y 136.365,Z 376.326,A -85,B 0,C 180,E1 -24886.185,E2 -24886.185} C_VEL
LIN {X 0,Y 137.045,Z 379.901,A -85,B 0,C 180,E1 -24892.025,E2 -24892.025} C_VEL
LIN {X 0,Y 137.169,Z 382.276,A -85,B 0,C 180,E1 -24895.7,E2 -24895.7} C_VEL
LIN {X 0,Y 136.394,Z 384.173,A -85,B 0,C 180,E1 -24898.503,E2 -24898.503} C_VEL
LIN {X 0,Y 137.543,Z 396.705,A -85,B 0,C 180,E1 -24900.306,E2 -24900.306} C_VEL
LIN {X 0,Y 138.162,Z 406.665,A -85,B 0,C 180,E1 -24902.223,E2 -24902.223} C_VEL
LIN {X 0,Y 138.358,Z 414.397,A -85,B 0,C 180,E1 -24904.021,E2 -24904.021} C_VEL
LIN {X 0,Y 138.437,Z 421.71,A -85,B 0,C 180,E1 -24906.042,E2 -24906.042} C_VEL
LIN {X 0,Y 138.274,Z 429.947,A -85,B 0,C 180,E1 -24908.773,E2 -24908.773} C_VEL
LIN {X 0,Y 138.017,Z 433.046,A -85,B 0,C 180,E1 -24909.901,E2 -24909.901} C_VEL
LIN {X 0,Y 136.227,Z 441.187,A -85,B 0,C 180,E1 -24913.52,E2 -24913.52} C_VEL
LIN {X 0,Y 135.158,Z 446.516,A -85,B 0,C 180,E1 -24916.472,E2 -24916.472} C_VEL
LIN {X 0,Y 134.446,Z 450.969,A -85,B 0,C 180,E1 -24919.462,E2 -24919.462} C_VEL
LIN {X 0,Y 133.998,Z 454.662,A -85,B 0,C 180,E1 -24922.47,E2 -24922.47} C_VEL
LIN {X 0,Y 133.879,Z 458.834,A -85,B 0,C 180,E1 -24926.995,E2 -24926.995} C_VEL
LIN {X 0,Y 134.032,Z 460.934,A -85,B 0,C 180,E1 -24930.004,E2 -24930.004} C_VEL
LIN {X 0,Y 133.723,Z 462.398,A -85,B 0,C 180,E1 -24933.017,E2 -24933.017} C_VEL
LIN {X 0,Y 133.712,Z 463.291,A -85,B 0,C 180,E1 -24936.038,E2 -24936.038} C_VEL
LIN {X 0,Y 134.009,Z 463.745,A -85,B 0,C 180,E1 -24939.056,E2 -24939.056} C_VEL
LIN {X 0,Y 134.658,Z 463.776,A -85,B 0,C 180,E1 -24942.054,E2 -24942.054} C_VEL
LIN {X 0,Y 135.661,Z 463.335,A -85,B 0,C 180,E1 -24945.016,E2 -24945.016} C_VEL
LIN {X 0,Y 137.036,Z 462.338,A -85,B 0,C 180,E1 -24947.925,E2 -24947.925} C_VEL
LIN {X 0,Y 138.744,Z 460.904,A -85,B 0,C 180,E1 -24950.772,E2 -24950.772} C_VEL
LIN {X 0,Y 142.171,Z 457.844,A -85,B 0,C 180,E1 -24954.85,E2 -24954.85} C_VEL
LIN {X 0,Y 146.333,Z 453.586,A -85,B 0,C 180,E1 -24958.707,E2 -24958.707} C_VEL
LIN {X 0,Y 149.387,Z 449.918,A -85,B 0,C 180,E1 -24961.169,E2 -24961.169} C_VEL
LIN {X 0,Y 152.633,Z 444.567,A -85,B 0,C 180,E1 -24964.34,E2 -24964.34} C_VEL
LIN {X 0,Y 155.334,Z 438.242,A -85,B 0,C 180,E1 -24967.651,E2 -24967.651} C_VEL
LIN {X 0,Y 157.572,Z 430.653,A -85,B 0,C 180,E1 -24971.209,E2 -24971.209} C_VEL
LIN {X 0,Y 158.293,Z 426.414,A -85,B 0,C 180,E1 -24973.14,E2 -24973.14} C_VEL
LIN {X 0,Y 158.051,Z 422.575,A -85,B 0,C 180,E1 -24975.358,E2 -24975.358} C_VEL
LIN {X 0,Y 157.224,Z 418.642,A -85,B 0,C 180,E1 -24977.891,E2 -24977.891} C_VEL
LIN {X 0,Y 156.235,Z 414.432,A -85,B 0,C 180,E1 -24980.964,E2 -24980.964} C_VEL
LIN {X 0,Y 155.252,Z 410.591,A -85,B 0,C 180,E1 -24983.947,E2 -24983.947} C_VEL
LIN {X 0,Y 153.955,Z 406.398,A -85,B 0,C 180,E1 -24988.243,E2 -24988.243} C_VEL
LIN {X 0,Y 153.215,Z 404.621,A -85,B 0,C 180,E1 -24990.643,E2 -24990.643} C_VEL
LIN {X 0,Y 152.001,Z 402.147,A -85,B 0,C 180,E1 -24996.044,E2 -24996.044} C_VEL
LIN {X 0,Y 151.838,Z 400.884,A -85,B 0,C 180,E1 -25001.092,E2 -25001.092} C_VEL
LIN {X 0,Y 152.458,Z 401.275,A -85,B 0,C 180,E1 -25006.672,E2 -25006.672} C_VEL
LIN {X 0,Y 152.639,Z 401.441,A -85,B 0,C 180,E1 -25007.422,E2 -25007.422} C_VEL
LIN {X 0,Y 152.984,Z 402.602,A -85,B 0,C 180,E1 -25009.585,E2 -25009.585} C_VEL
LIN {X 0,Y 152.823,Z 404.748,A -85,B 0,C 180,E1 -25011.658,E2 -25011.658} C_VEL
LIN {X 0,Y 152.02,Z 412.034,A -85,B 0,C 180,E1 -25017.068,E2 -25017.068} C_VEL
LIN {X 0,Y 152.106,Z 413.557,A -85,B 0,C 180,E1 -25018.479,E2 -25018.479} C_VEL
LIN {X 0,Y 153.072,Z 417.971,A -85,B 0,C 180,E1 -25022.629,E2 -25022.629} C_VEL
LIN {X 0,Y 153.662,Z 422.805,A -85,B 0,C 180,E1 -25026.563,E2 -25026.563} C_VEL
LIN {X 0,Y 153.373,Z 427.485,A -85,B 0,C 180,E1 -25029.892,E2 -25029.892} C_VEL
LIN {X 0,Y 152.106,Z 432.721,A -85,B 0,C 180,E1 -25033.354,E2 -25033.354} C_VEL
LIN {X 0,Y 151.06,Z 435.096,A -85,B 0,C 180,E1 -25034.822,E2 -25034.822} C_VEL
LIN {X 0,Y 146.204,Z 440.75,A -85,B 0,C 180,E1 -25038.065,E2 -25038.065} C_VEL
LIN {X 0,Y 142.693,Z 444.251,A -85,B 0,C 180,E1 -25040.633,E2 -25040.633} C_VEL
LIN {X 0,Y 138.645,Z 447.748,A -85,B 0,C 180,E1 -25044.148,E2 -25044.148} C_VEL
LIN {X 0,Y 135.101,Z 450.282,A -85,B 0,C 180,E1 -25047.913,E2 -25047.913} C_VEL
LIN {X 0,Y 131.883,Z 451.984,A -85,B 0,C 180,E1 -25052.197,E2 -25052.197} C_VEL
LIN {X 0,Y 129.416,Z 452.63,A -85,B 0,C 180,E1 -25056.677,E2 -25056.677} C_VEL
LIN {X 0,Y 127.594,Z 452.22,A -85,B 0,C 180,E1 -25061.369,E2 -25061.369} C_VEL
LIN {X 0,Y 126.518,Z 450.638,A -85,B 0,C 180,E1 -25066.226,E2 -25066.226} C_VEL
LIN {X 0,Y 126.311,Z 446.972,A -85,B 0,C 180,E1 -25072.258,E2 -25072.258} C_VEL
LIN {X 0,Y 126.73,Z 443.423,A -85,B 0,C 180,E1 -25076.315,E2 -25076.315} C_VEL
LIN {X 0,Y 127.609,Z 438.908,A -85,B 0,C 180,E1 -25080.282,E2 -25080.282} C_VEL
LIN {X 0,Y 129.097,Z 432.149,A -85,B 0,C 180,E1 -25084.86,E2 -25084.86} C_VEL
LIN {X 0,Y 130.91,Z 424.49,A -85,B 0,C 180,E1 -25088.75,E2 -25088.75} C_VEL
LIN {X 0,Y 132.33,Z 418.02,A -85,B 0,C 180,E1 -25091.414,E2 -25091.414} C_VEL
LIN {X 0,Y 134.155,Z 410.149,A -85,B 0,C 180,E1 -25094.032,E2 -25094.032} C_VEL
LIN {X 0,Y 133.777,Z 403.995,A -85,B 0,C 180,E1 -25095.934,E2 -25095.934} C_VEL
LIN {X 0,Y 132.874,Z 395.979,A -85,B 0,C 180,E1 -25098.094,E2 -25098.094} C_VEL
LIN {X 0,Y 131.785,Z 388.29,A -85,B 0,C 180,E1 -25099.873,E2 -25099.873} C_VEL
LIN {X 0,Y 129.623,Z 379.308,A -85,B 0,C 180,E1 -25101.716,E2 -25101.716} C_VEL
LIN {X 0,Y 129.041,Z 377.227,A -85,B 0,C 180,E1 -25102.17,E2 -25102.17} C_VEL
LIN {X 0,Y 129.582,Z 377.159,A -85,B 0,C 180,E1 -25106.887,E2 -25106.887} C_VEL
LIN {X 0,Y 130.067,Z 377.098,A -85,B 0,C 180,E1 -25109.996,E2 -25109.996} C_VEL
LIN {X 0,Y 129.522,Z 377.163,A -85,B 0,C 180,E1 -25119.364,E2 -25119.364} C_VEL
LIN {X 0,Y 129.385,Z 377.177,A -85,B 0,C 180,E1 -25122.545,E2 -25122.545} C_VEL
LIN {X 0,Y 129.15,Z 377.206,A -85,B 0,C 180,E1 -25129.052,E2 -25129.052} C_VEL
LIN {X 0,Y 129.098,Z 377.215,A -85,B 0,C 180,E1 -25132.396,E2 -25132.396} C_VEL
LIN {X 0,Y 129.025,Z 377.221,A -85,B 0,C 180,E1 -25139.371,E2 -25139.371} C_VEL
LIN {X 0,Y 129.017,Z 377.222,A -85,B 0,C 180,E1 -25145.211,E2 -25145.211} C_VEL
LIN {X 0,Y 129.039,Z 377.224,A -85,B 0,C 180,E1 -25150.806,E2 -25150.806} C_VEL
LIN {X 0,Y 129.028,Z 377.22,A -85,B 0,C 180,E1 -25155.074,E2 -25155.074} C_VEL
LIN {X 0,Y 129.038,Z 377.223,A -85,B 0,C 180,E1 -25159.679,E2 -25159.679} C_VEL
LIN {X 0,Y 129.016,Z 377.224,A -85,B 0,C 180,E1 -25164.789,E2 -25164.789} C_VEL
LIN {X 0,Y 129.022,Z 377.221,A -85,B 0,C 180,E1 -25170.647,E2 -25170.647} C_VEL
LIN {X 0,Y 129.125,Z 377.211,A -85,B 0,C 180,E1 -25177.608,E2 -25177.608} C_VEL
LIN {X 0,Y 129.176,Z 377.204,A -85,B 0,C 180,E1 -25180.951,E2 -25180.951} C_VEL
LIN {X 0,Y 129.408,Z 377.172,A -85,B 0,C 180,E1 -25187.817,E2 -25187.817} C_VEL
LIN {X 0,Y 129.52,Z 377.164,A -85,B 0,C 180,E1 -25190.635,E2 -25190.635} C_VEL
LIN {X 0,Y 130.081,Z 377.095,A -85,B 0,C 180,E1 -25200.003,E2 -25200.003} C_VEL
LIN {X 0,Y 129.515,Z 377.165,A -85,B 0,C 180,E1 -25209.372,E2 -25209.372} C_VEL
LIN {X 0,Y 129.385,Z 377.173,A -85,B 0,C 180,E1 -25212.552,E2 -25212.552} C_VEL
LIN {X 0,Y 129.151,Z 377.209,A -85,B 0,C 180,E1 -25219.06,E2 -25219.06} C_VEL
LIN {X 0,Y 129.102,Z 377.212,A -85,B 0,C 180,E1 -25222.403,E2 -25222.403} C_VEL
LIN {X 0,Y 129.025,Z 377.225,A -85,B 0,C 180,E1 -25225.837,E2 -25225.837} C_VEL
LIN {X 0,Y 129.011,Z 377.222,A -85,B 0,C 180,E1 -25229.362,E2 -25229.362} C_VEL
LIN {X 0,Y 128.977,Z 377.23,A -85,B 0,C 180,E1 -25235.187,E2 -25235.187} C_VEL
LIN {X 0,Y 128.986,Z 377.23,A -85,B 0,C 180,E1 -25240.835,E2 -25240.835} C_VEL
LIN {X 0,Y 129.356,Z 377.365,A -85,B 0,C 180,E1 -25246.61,E2 -25246.61} C_VEL
LIN {X 0,Y 129.926,Z 380.226,A -85,B 0,C 180,E1 -25251.539,E2 -25251.539} C_VEL
LIN {X 0,Y 130.067,Z 381.807,A -85,B 0,C 180,E1 -25254.15,E2 -25254.15} C_VEL
LIN {X 0,Y 129.54,Z 383.931,A -85,B 0,C 180,E1 -25257.394,E2 -25257.394} C_VEL
LIN {X 0,Y 130.69,Z 396.747,A -85,B 0,C 180,E1 -25259.369,E2 -25259.369} C_VEL
LIN {X 0,Y 131.201,Z 405.721,A -85,B 0,C 180,E1 -25261.182,E2 -25261.182} C_VEL
LIN {X 0,Y 131.409,Z 414.689,A -85,B 0,C 180,E1 -25263.395,E2 -25263.395} C_VEL
LIN {X 0,Y 131.438,Z 422.522,A -85,B 0,C 180,E1 -25265.729,E2 -25265.729} C_VEL
LIN {X 0,Y 131.22,Z 430.043,A -85,B 0,C 180,E1 -25268.399,E2 -25268.399} C_VEL
LIN {X 0,Y 130.922,Z 433.102,A -85,B 0,C 180,E1 -25269.583,E2 -25269.583} C_VEL
LIN {X 0,Y 129.119,Z 441.151,A -85,B 0,C 180,E1 -25273.4,E2 -25273.4} C_VEL
LIN {X 0,Y 128.025,Z 446.424,A -85,B 0,C 180,E1 -25276.513,E2 -25276.513} C_VEL
LIN {X 0,Y 127.195,Z 451.774,A -85,B 0,C 180,E1 -25280.463,E2 -25280.463} C_VEL
LIN {X 0,Y 126.819,Z 456.31,A -85,B 0,C 180,E1 -25284.796,E2 -25284.796} C_VEL
LIN {X 0,Y 126.83,Z 459.052,A -85,B 0,C 180,E1 -25288.262,E2 -25288.262} C_VEL
LIN {X 0,Y 126.967,Z 460.251,A -85,B 0,C 180,E1 -25290.004,E2 -25290.004} C_VEL
LIN {X 0,Y 126.665,Z 461.749,A -85,B 0,C 180,E1 -25293.185,E2 -25293.185} C_VEL
LIN {X 0,Y 126.672,Z 462.761,A -85,B 0,C 180,E1 -25296.375,E2 -25296.375} C_VEL
LIN {X 0,Y 126.999,Z 463.339,A -85,B 0,C 180,E1 -25299.56,E2 -25299.56} C_VEL
LIN {X 0,Y 127.704,Z 463.488,A -85,B 0,C 180,E1 -25302.721,E2 -25302.721} C_VEL
LIN {X 0,Y 128.792,Z 463.071,A -85,B 0,C 180,E1 -25305.838,E2 -25305.838} C_VEL
LIN {X 0,Y 130.271,Z 462.203,A -85,B 0,C 180,E1 -25308.891,E2 -25308.891} C_VEL
LIN {X 0,Y 132.119,Z 460.91,A -85,B 0,C 180,E1 -25311.865,E2 -25311.865} C_VEL
LIN {X 0,Y 135.751,Z 457.993,A -85,B 0,C 180,E1 -25316.111,E2 -25316.111} C_VEL
LIN {X 0,Y 140.159,Z 453.918,A -85,B 0,C 180,E1 -25320.099,E2 -25320.099} C_VEL
LIN {X 0,Y 143.344,Z 450.45,A -85,B 0,C 180,E1 -25322.641,E2 -25322.641} C_VEL
LIN {X 0,Y 146.137,Z 446.426,A -85,B 0,C 180,E1 -25325.251,E2 -25325.251} C_VEL
LIN {X 0,Y 148.601,Z 441.813,A -85,B 0,C 180,E1 -25327.944,E2 -25327.944} C_VEL
LIN {X 0,Y 151.109,Z 435.491,A -85,B 0,C 180,E1 -25331.288,E2 -25331.288} C_VEL
LIN {X 0,Y 152.559,Z 430.722,A -85,B 0,C 180,E1 -25333.714,E2 -25333.714} C_VEL
LIN {X 0,Y 152.776,Z 428.222,A -85,B 0,C 180,E1 -25335.112,E2 -25335.112} C_VEL
LIN {X 0,Y 152.315,Z 423.725,A -85,B 0,C 180,E1 -25338.271,E2 -25338.271} C_VEL
LIN {X 0,Y 151.36,Z 418.849,A -85,B 0,C 180,E1 -25342.13,E2 -25342.13} C_VEL
LIN {X 0,Y 150.88,Z 415.856,A -85,B 0,C 180,E1 -25344.769,E2 -25344.769} C_VEL
LIN {X 0,Y 149.922,Z 411.962,A -85,B 0,C 180,E1 -25348.956,E2 -25348.956} C_VEL
LIN {X 0,Y 148.853,Z 409.281,A -85,B 0,C 180,E1 -25353.783,E2 -25353.783} C_VEL
LIN {X 0,Y 148.466,Z 407.863,A -85,B 0,C 180,E1 -25357.744,E2 -25357.744} C_VEL
LIN {X 0,Y 148.486,Z 407.119,A -85,B 0,C 180,E1 -25361.205,E2 -25361.205} C_VEL
LIN {X 0,Y 149.133,Z 407.603,A -85,B 0,C 180,E1 -25367.368,E2 -25367.368} C_VEL
LIN {X 0,Y 149.821,Z 408.277,A -85,B 0,C 180,E1 -25370.111,E2 -25370.111} C_VEL
LIN {X 0,Y 150.352,Z 408.944,A -85,B 0,C 180,E1 -25371.936,E2 -25371.936} C_VEL
LIN {X 0,Y 151.906,Z 412.482,A -85,B 0,C 180,E1 -25377.346,E2 -25377.346} C_VEL
LIN {X 0,Y 152.106,Z 413.557,A -85,B 0,C 180,E1 -25378.479,E2 -25378.479} C_VEL
LIN {X 0,Y 152.243,Z 416.104,A -85,B 0,C 180,E1 -25380.507,E2 -25380.507} C_VEL
LIN {X 0,Y 151.463,Z 419.363,A -85,B 0,C 180,E1 -25382.382,E2 -25382.382} C_VEL
LIN {X 0,Y 148.959,Z 426.308,A -85,B 0,C 180,E1 -25386.04,E2 -25386.04} C_VEL
LIN {X 0,Y 147.607,Z 430.359,A -85,B 0,C 180,E1 -25388.682,E2 -25388.682} C_VEL
LIN {X 0,Y 146.045,Z 435.326,A -85,B 0,C 180,E1 -25392.347,E2 -25392.347} C_VEL
LIN {X 0,Y 144.705,Z 437.381,A -85,B 0,C 180,E1 -25393.734,E2 -25393.734} C_VEL
LIN {X 0,Y 139.651,Z 442.619,A -85,B 0,C 180,E1 -25397.013,E2 -25397.013} C_VEL
LIN {X 0,Y 133.75,Z 447.647,A -85,B 0,C 180,E1 -25401.578,E2 -25401.578} C_VEL
LIN {X 0,Y 129.479,Z 450.493,A -85,B 0,C 180,E1 -25405.733,E2 -25405.733} C_VEL
LIN {X 0,Y 127.473,Z 451.649,A -85,B 0,C 180,E1 -25408.091,E2 -25408.091} C_VEL
LIN {X 0,Y 124.555,Z 452.769,A -85,B 0,C 180,E1 -25412.174,E2 -25412.174} C_VEL
LIN {X 0,Y 122.287,Z 453.036,A -85,B 0,C 180,E1 -25416.422,E2 -25416.422} C_VEL
LIN {X 0,Y 120.633,Z 452.461,A -85,B 0,C 180,E1 -25420.761,E2 -25420.761} C_VEL
LIN {X 0,Y 119.567,Z 451.056,A -85,B 0,C 180,E1 -25425.137,E2 -25425.137} C_VEL
LIN {X 0,Y 119.139,Z 448.436,A -85,B 0,C 180,E1 -25430.068,E2 -25430.068} C_VEL
LIN {X 0,Y 119.477,Z 444.262,A -85,B 0,C 180,E1 -25435.432,E2 -25435.432} C_VEL
LIN {X 0,Y 120.285,Z 439.86,A -85,B 0,C 180,E1 -25439.661,E2 -25439.661} C_VEL
LIN {X 0,Y 121.709,Z 433.603,A -85,B 0,C 180,E1 -25444.332,E2 -25444.332} C_VEL
LIN {X 0,Y 123.619,Z 425.734,A -85,B 0,C 180,E1 -25448.746,E2 -25448.746} C_VEL
LIN {X 0,Y 125.47,Z 417.784,A -85,B 0,C 180,E1 -25452.206,E2 -25452.206} C_VEL
LIN {X 0,Y 127.274,Z 410.346,A -85,B 0,C 180,E1 -25454.79,E2 -25454.79} C_VEL
LIN {X 0,Y 126.707,Z 402.916,A -85,B 0,C 180,E1 -25457.177,E2 -25457.177} C_VEL
LIN {X 0,Y 125.696,Z 394.398,A -85,B 0,C 180,E1 -25459.526,E2 -25459.526} C_VEL
LIN {X 0,Y 124.709,Z 387.871,A -85,B 0,C 180,E1 -25461.08,E2 -25461.08} C_VEL
LIN {X 0,Y 122.49,Z 379.792,A -85,B 0,C 180,E1 -25462.889,E2 -25462.889} C_VEL
LIN {X 0,Y 122.112,Z 378.09,A -85,B 0,C 180,E1 -25463.282,E2 -25463.282} C_VEL
LIN {X 0,Y 123.016,Z 377.977,A -85,B 0,C 180,E1 -25469.996,E2 -25469.996} C_VEL
LIN {X 0,Y 122.448,Z 378.044,A -85,B 0,C 180,E1 -25476.587,E2 -25476.587} C_VEL
LIN {X 0,Y 122.448,Z 378.042,A -85,B 0,C 180,E1 -25479.911,E2 -25479.911} C_VEL
LIN {X 0,Y 122.255,Z 378.065,A -85,B 0,C 180,E1 -25483.289,E2 -25483.289} C_VEL
LIN {X 0,Y 122.039,Z 378.09,A -85,B 0,C 180,E1 -25490.209,E2 -25490.209} C_VEL
LIN {X 0,Y 121.973,Z 378.105,A -85,B 0,C 180,E1 -25493.782,E2 -25493.782} C_VEL
LIN {X 0,Y 121.931,Z 378.107,A -85,B 0,C 180,E1 -25500.172,E2 -25500.172} C_VEL
LIN {X 0,Y 121.939,Z 378.101,A -85,B 0,C 180,E1 -25506.213,E2 -25506.213} C_VEL
LIN {X 0,Y 121.958,Z 378.105,A -85,B 0,C 180,E1 -25511.49,E2 -25511.49} C_VEL
LIN {X 0,Y 121.957,Z 378.106,A -85,B 0,C 180,E1 -25518.51,E2 -25518.51} C_VEL
LIN {X 0,Y 121.967,Z 378.102,A -85,B 0,C 180,E1 -25524.819,E2 -25524.819} C_VEL
LIN {X 0,Y 121.93,Z 378.106,A -85,B 0,C 180,E1 -25529.827,E2 -25529.827} C_VEL
LIN {X 0,Y 122.057,Z 378.092,A -85,B 0,C 180,E1 -25537.101,E2 -25537.101} C_VEL
LIN {X 0,Y 122.122,Z 378.085,A -85,B 0,C 180,E1 -25543.281,E2 -25543.281} C_VEL
LIN {X 0,Y 122.355,Z 378.05,A -85,B 0,C 180,E1 -25547.524,E2 -25547.524} C_VEL
LIN {X 0,Y 122.447,Z 378.043,A -85,B 0,C 180,E1 -25550.088,E2 -25550.088} C_VEL
LIN {X 0,Y 122.6,Z 378.021,A -85,B 0,C 180,E1 -25556.717,E2 -25556.717} C_VEL
LIN {X 0,Y 123.035,Z 377.973,A -85,B 0,C 180,E1 -25560.003,E2 -25560.003} C_VEL
LIN {X 0,Y 122.444,Z 378.044,A -85,B 0,C 180,E1 -25566.595,E2 -25566.595} C_VEL
LIN {X 0,Y 122.443,Z 378.044,A -85,B 0,C 180,E1 -25569.919,E2 -25569.919} C_VEL
LIN {X 0,Y 122.255,Z 378.062,A -85,B 0,C 180,E1 -25573.297,E2 -25573.297} C_VEL
LIN {X 0,Y 122.041,Z 378.09,A -85,B 0,C 180,E1 -25580.217,E2 -25580.217} C_VEL
LIN {X 0,Y 121.978,Z 378.103,A -85,B 0,C 180,E1 -25583.789,E2 -25583.789} C_VEL
LIN {X 0,Y 121.924,Z 378.106,A -85,B 0,C 180,E1 -25590.168,E2 -25590.168} C_VEL
LIN {X 0,Y 121.895,Z 378.11,A -85,B 0,C 180,E1 -25596.186,E2 -25596.186} C_VEL
LIN {X 0,Y 122.043,Z 378.093,A -85,B 0,C 180,E1 -25603.716,E2 -25603.716} C_VEL
LIN {X 0,Y 122.31,Z 378.163,A -85,B 0,C 180,E1 -25606.667,E2 -25606.667} C_VEL
LIN {X 0,Y 122.78,Z 380.527,A -85,B 0,C 180,E1 -25610.982,E2 -25610.982} C_VEL
LIN {X 0,Y 122.918,Z 381.781,A -85,B 0,C 180,E1 -25613.18,E2 -25613.18} C_VEL
LIN {X 0,Y 122.618,Z 383.527,A -85,B 0,C 180,E1 -25616.148,E2 -25616.148} C_VEL
LIN {X 0,Y 123.737,Z 395.432,A -85,B 0,C 180,E1 -25618.069,E2 -25618.069} C_VEL
LIN {X 0,Y 124.325,Z 406.125,A -85,B 0,C 180,E1 -25620.36,E2 -25620.36} C_VEL
LIN {X 0,Y 124.486,Z 414.983,A -85,B 0,C 180,E1 -25622.701,E2 -25622.701} C_VEL
LIN {X 0,Y 124.423,Z 423.668,A -85,B 0,C 180,E1 -25625.495,E2 -25625.495} C_VEL
LIN {X 0,Y 124.144,Z 431.196,A -85,B 0,C 180,E1 -25628.414,E2 -25628.414} C_VEL
LIN {X 0,Y 122.639,Z 438.181,A -85,B 0,C 180,E1 -25631.633,E2 -25631.633} C_VEL
LIN {X 0,Y 121.124,Z 445.171,A -85,B 0,C 180,E1 -25635.728,E2 -25635.728} C_VEL
LIN {X 0,Y 120.191,Z 450.684,A -85,B 0,C 180,E1 -25639.901,E2 -25639.901} C_VEL
LIN {X 0,Y 119.802,Z 454.287,A -85,B 0,C 180,E1 -25643.267,E2 -25643.267} C_VEL
LIN {X 0,Y 119.776,Z 457.225,A -85,B 0,C 180,E1 -25646.641,E2 -25646.641} C_VEL
LIN {X 0,Y 119.904,Z 459.463,A -85,B 0,C 180,E1 -25650.004,E2 -25650.004} C_VEL
LIN {X 0,Y 119.598,Z 461.069,A -85,B 0,C 180,E1 -25653.373,E2 -25653.373} C_VEL
LIN {X 0,Y 119.626,Z 462.216,A -85,B 0,C 180,E1 -25656.752,E2 -25656.752} C_VEL
LIN {X 0,Y 119.991,Z 462.931,A -85,B 0,C 180,E1 -25660.124,E2 -25660.124} C_VEL
LIN {X 0,Y 120.779,Z 463.117,A -85,B 0,C 180,E1 -25663.464,E2 -25663.464} C_VEL
LIN {X 0,Y 121.96,Z 462.799,A -85,B 0,C 180,E1 -25666.75,E2 -25666.75} C_VEL
LIN {X 0,Y 123.548,Z 462.071,A -85,B 0,C 180,E1 -25669.961,E2 -25669.961} C_VEL
LIN {X 0,Y 125.553,Z 460.93,A -85,B 0,C 180,E1 -25673.073,E2 -25673.073} C_VEL
LIN {X 0,Y 129.411,Z 458.188,A -85,B 0,C 180,E1 -25677.496,E2 -25677.496} C_VEL
LIN {X 0,Y 134.079,Z 454.28,A -85,B 0,C 180,E1 -25681.616,E2 -25681.616} C_VEL
LIN {X 0,Y 137.416,Z 450.994,A -85,B 0,C 180,E1 -25684.239,E2 -25684.239} C_VEL
LIN {X 0,Y 141.045,Z 446.064,A -85,B 0,C 180,E1 -25687.622,E2 -25687.622} C_VEL
LIN {X 0,Y 144.181,Z 440.29,A -85,B 0,C 180,E1 -25691.156,E2 -25691.156} C_VEL
LIN {X 0,Y 146.504,Z 434.663,A -85,B 0,C 180,E1 -25694.316,E2 -25694.316} C_VEL
LIN {X 0,Y 147.1,Z 432.194,A -85,B 0,C 180,E1 -25695.783,E2 -25695.783} C_VEL
LIN {X 0,Y 147.013,Z 427.993,A -85,B 0,C 180,E1 -25699.022,E2 -25699.022} C_VEL
LIN {X 0,Y 146.446,Z 423.367,A -85,B 0,C 180,E1 -25703.138,E2 -25703.138} C_VEL
LIN {X 0,Y 146.316,Z 421.622,A -85,B 0,C 180,E1 -25704.8,E2 -25704.8} C_VEL
LIN {X 0,Y 145.478,Z 416.941,A -85,B 0,C 180,E1 -25710.416,E2 -25710.416} C_VEL
LIN {X 0,Y 144.908,Z 415.11,A -85,B 0,C 180,E1 -25714.117,E2 -25714.117} C_VEL
LIN {X 0,Y 144.647,Z 413.383,A -85,B 0,C 180,E1 -25720.114,E2 -25720.114} C_VEL
LIN {X 0,Y 144.788,Z 413.153,A -85,B 0,C 180,E1 -25723.065,E2 -25723.065} C_VEL
LIN {X 0,Y 145.584,Z 413.784,A -85,B 0,C 180,E1 -25728.864,E2 -25728.864} C_VEL
LIN {X 0,Y 146.198,Z 414.684,A -85,B 0,C 180,E1 -25731.706,E2 -25731.706} C_VEL
LIN {X 0,Y 147.391,Z 418.124,A -85,B 0,C 180,E1 -25737.264,E2 -25737.264} C_VEL
LIN {X 0,Y 147.99,Z 423.332,A -85,B 0,C 180,E1 -25742.719,E2 -25742.719} C_VEL
LIN {X 0,Y 148.061,Z 426.252,A -85,B 0,C 180,E1 -25745.445,E2 -25745.445} C_VEL
LIN {X 0,Y 147.607,Z 430.359,A -85,B 0,C 180,E1 -25748.682,E2 -25748.682} C_VEL
LIN {X 0,Y 146.481,Z 432.448,A -85,B 0,C 180,E1 -25749.9,E2 -25749.9} C_VEL
LIN {X 0,Y 143.602,Z 435.61,A -85,B 0,C 180,E1 -25751.172,E2 -25751.172} C_VEL
LIN {X 0,Y 137.33,Z 440.783,A -85,B 0,C 180,E1 -25753.289,E2 -25753.289} C_VEL
LIN {X 0,Y 135.824,Z 442.043,A -85,B 0,C 180,E1 -25754.087,E2 -25754.087} C_VEL
LIN {X 0,Y 130.211,Z 446.709,A -85,B 0,C 180,E1 -25757.975,E2 -25757.975} C_VEL
LIN {X 0,Y 125.57,Z 449.889,A -85,B 0,C 180,E1 -25761.925,E2 -25761.925} C_VEL
LIN {X 0,Y 120.068,Z 452.534,A -85,B 0,C 180,E1 -25767.918,E2 -25767.918} C_VEL
LIN {X 0,Y 116.868,Z 453.309,A -85,B 0,C 180,E1 -25772.763,E2 -25772.763} C_VEL
LIN {X 0,Y 114.416,Z 453.04,A -85,B 0,C 180,E1 -25777.893,E2 -25777.893} C_VEL
LIN {X 0,Y 112.836,Z 451.691,A -85,B 0,C 180,E1 -25783.241,E2 -25783.241} C_VEL
LIN {X 0,Y 112.092,Z 449.114,A -85,B 0,C 180,E1 -25788.791,E2 -25788.791} C_VEL
LIN {X 0,Y 112.259,Z 445.07,A -85,B 0,C 180,E1 -25794.469,E2 -25794.469} C_VEL
LIN {X 0,Y 113.042,Z 440.606,A -85,B 0,C 180,E1 -25799.137,E2 -25799.137} C_VEL
LIN {X 0,Y 113.926,Z 436.672,A -85,B 0,C 180,E1 -25802.451,E2 -25802.451} C_VEL
LIN {X 0,Y 115.207,Z 431.234,A -85,B 0,C 180,E1 -25806.202,E2 -25806.202} C_VEL
LIN {X 0,Y 116.808,Z 424.998,A -85,B 0,C 180,E1 -25809.683,E2 -25809.683} C_VEL
LIN {X 0,Y 118.413,Z 418.309,A -85,B 0,C 180,E1 -25812.733,E2 -25812.733} C_VEL
LIN {X 0,Y 120.323,Z 410.438,A -85,B 0,C 180,E1 -25815.622,E2 -25815.622} C_VEL
LIN {X 0,Y 119.602,Z 401.747,A -85,B 0,C 180,E1 -25818.557,E2 -25818.557} C_VEL
LIN {X 0,Y 118.376,Z 391.475,A -85,B 0,C 180,E1 -25821.46,E2 -25821.46} C_VEL
LIN {X 0,Y 115.888,Z 381.563,A -85,B 0,C 180,E1 -25823.903,E2 -25823.903} C_VEL
LIN {X 0,Y 115.164,Z 378.956,A -85,B 0,C 180,E1 -25824.524,E2 -25824.524} C_VEL
LIN {X 0,Y 115.961,Z 378.856,A -85,B 0,C 180,E1 -25829.996,E2 -25829.996} C_VEL
LIN {X 0,Y 115.389,Z 378.923,A -85,B 0,C 180,E1 -25836.992,E2 -25836.992} C_VEL
LIN {X 0,Y 115.384,Z 378.92,A -85,B 0,C 180,E1 -25840.524,E2 -25840.524} C_VEL
LIN {X 0,Y 115.139,Z 378.955,A -85,B 0,C 180,E1 -25844.127,E2 -25844.127} C_VEL
LIN {X 0,Y 114.971,Z 378.972,A -85,B 0,C 180,E1 -25851.512,E2 -25851.512} C_VEL
LIN {X 0,Y 114.86,Z 378.99,A -85,B 0,C 180,E1 -25855.355,E2 -25855.355} C_VEL
LIN {X 0,Y 114.858,Z 378.989,A -85,B 0,C 180,E1 -25861.066,E2 -25861.066} C_VEL
LIN {X 0,Y 114.871,Z 378.985,A -85,B 0,C 180,E1 -25867.715,E2 -25867.715} C_VEL
LIN {X 0,Y 114.876,Z 378.986,A -85,B 0,C 180,E1 -25872.77,E2 -25872.77} C_VEL
LIN {X 0,Y 114.882,Z 378.987,A -85,B 0,C 180,E1 -25877.711,E2 -25877.711} C_VEL
LIN {X 0,Y 114.874,Z 378.982,A -85,B 0,C 180,E1 -25882.679,E2 -25882.679} C_VEL
LIN {X 0,Y 114.858,Z 378.988,A -85,B 0,C 180,E1 -25888.932,E2 -25888.932} C_VEL
LIN {X 0,Y 114.955,Z 378.978,A -85,B 0,C 180,E1 -25896.486,E2 -25896.486} C_VEL
LIN {X 0,Y 115.024,Z 378.968,A -85,B 0,C 180,E1 -25902.215,E2 -25902.215} C_VEL
LIN {X 0,Y 115.297,Z 378.93,A -85,B 0,C 180,E1 -25907.213,E2 -25907.213} C_VEL
LIN {X 0,Y 115.387,Z 378.923,A -85,B 0,C 180,E1 -25913.007,E2 -25913.007} C_VEL
LIN {X 0,Y 115.987,Z 378.851,A -85,B 0,C 180,E1 -25920.003,E2 -25920.003} C_VEL
LIN {X 0,Y 115.386,Z 378.923,A -85,B 0,C 180,E1 -25927,E2 -25927} C_VEL
LIN {X 0,Y 115.277,Z 378.93,A -85,B 0,C 180,E1 -25932.743,E2 -25932.743} C_VEL
LIN {X 0,Y 115.008,Z 378.971,A -85,B 0,C 180,E1 -25937.794,E2 -25937.794} C_VEL
LIN {X 0,Y 114.942,Z 378.979,A -85,B 0,C 180,E1 -25943.498,E2 -25943.498} C_VEL
LIN {X 0,Y 114.857,Z 378.987,A -85,B 0,C 180,E1 -25951.068,E2 -25951.068} C_VEL
LIN {X 0,Y 114.798,Z 378.991,A -85,B 0,C 180,E1 -25957.753,E2 -25957.753} C_VEL
LIN {X 0,Y 115.185,Z 378.943,A -85,B 0,C 180,E1 -25965.869,E2 -25965.869} C_VEL
LIN {X 0,Y 115.286,Z 379.094,A -85,B 0,C 180,E1 -25967.02,E2 -25967.02} C_VEL
LIN {X 0,Y 115.793,Z 382,A -85,B 0,C 180,E1 -25972.637,E2 -25972.637} C_VEL
LIN {X 0,Y 115.714,Z 383.394,A -85,B 0,C 180,E1 -25974.832,E2 -25974.832} C_VEL
LIN {X 0,Y 116.83,Z 393.283,A -85,B 0,C 180,E1 -25976.519,E2 -25976.519} C_VEL
LIN {X 0,Y 117.391,Z 404.265,A -85,B 0,C 180,E1 -25978.917,E2 -25978.917} C_VEL
LIN {X 0,Y 117.55,Z 413.476,A -85,B 0,C 180,E1 -25981.431,E2 -25981.431} C_VEL
LIN {X 0,Y 117.473,Z 422.2,A -85,B 0,C 180,E1 -25984.332,E2 -25984.332} C_VEL
LIN {X 0,Y 117.17,Z 430.144,A -85,B 0,C 180,E1 -25987.524,E2 -25987.524} C_VEL
LIN {X 0,Y 116.338,Z 434.764,A -85,B 0,C 180,E1 -25989.679,E2 -25989.679} C_VEL
LIN {X 0,Y 114.876,Z 440.986,A -85,B 0,C 180,E1 -25993.111,E2 -25993.111} C_VEL
LIN {X 0,Y 113.801,Z 446.163,A -85,B 0,C 180,E1 -25996.614,E2 -25996.614} C_VEL
LIN {X 0,Y 112.966,Z 451.412,A -85,B 0,C 180,E1 -26001.057,E2 -26001.057} C_VEL
LIN {X 0,Y 112.688,Z 454.788,A -85,B 0,C 180,E1 -26004.639,E2 -26004.639} C_VEL
LIN {X 0,Y 112.767,Z 457.833,A -85,B 0,C 180,E1 -26008.707,E2 -26008.707} C_VEL
LIN {X 0,Y 112.841,Z 458.634,A -85,B 0,C 180,E1 -26010.005,E2 -26010.005} C_VEL
LIN {X 0,Y 112.542,Z 460.386,A -85,B 0,C 180,E1 -26013.585,E2 -26013.585} C_VEL
LIN {X 0,Y 112.573,Z 461.67,A -85,B 0,C 180,E1 -26017.177,E2 -26017.177} C_VEL
LIN {X 0,Y 113.009,Z 462.467,A -85,B 0,C 180,E1 -26020.757,E2 -26020.757} C_VEL
LIN {X 0,Y 113.884,Z 462.706,A -85,B 0,C 180,E1 -26024.296,E2 -26024.296} C_VEL
LIN {X 0,Y 115.168,Z 462.534,A -85,B 0,C 180,E1 -26027.77,E2 -26027.77} C_VEL
LIN {X 0,Y 116.875,Z 461.957,A -85,B 0,C 180,E1 -26031.154,E2 -26031.154} C_VEL
LIN {X 0,Y 119.052,Z 460.9,A -85,B 0,C 180,E1 -26034.412,E2 -26034.412} C_VEL
LIN {X 0,Y 123.16,Z 458.379,A -85,B 0,C 180,E1 -26039.02,E2 -26039.02} C_VEL
LIN {X 0,Y 128.091,Z 454.648,A -85,B 0,C 180,E1 -26043.28,E2 -26043.28} C_VEL
LIN {X 0,Y 132.498,Z 450.552,A -85,B 0,C 180,E1 -26046.737,E2 -26046.737} C_VEL
LIN {X 0,Y 136.126,Z 445.817,A -85,B 0,C 180,E1 -26050.197,E2 -26050.197} C_VEL
LIN {X 0,Y 139.432,Z 440.118,A -85,B 0,C 180,E1 -26053.878,E2 -26053.878} C_VEL
LIN {X 0,Y 141.24,Z 436.268,A -85,B 0,C 180,E1 -26056.301,E2 -26056.301} C_VEL
LIN {X 0,Y 141.505,Z 433.888,A -85,B 0,C 180,E1 -26058.163,E2 -26058.163} C_VEL
LIN {X 0,Y 141.443,Z 429.113,A -85,B 0,C 180,E1 -26062.661,E2 -26062.661} C_VEL
LIN {X 0,Y 141.156,Z 425.311,A -85,B 0,C 180,E1 -26066.789,E2 -26066.789} C_VEL
LIN {X 0,Y 140.967,Z 422.87,A -85,B 0,C 180,E1 -26070.093,E2 -26070.093} C_VEL
LIN {X 0,Y 140.614,Z 420.82,A -85,B 0,C 180,E1 -26074.12,E2 -26074.12} C_VEL
LIN {X 0,Y 140.405,Z 419.244,A -85,B 0,C 180,E1 -26079.486,E2 -26079.486} C_VEL
LIN {X 0,Y 140.51,Z 418.91,A -85,B 0,C 180,E1 -26082.533,E2 -26082.533} C_VEL
LIN {X 0,Y 141.219,Z 419.378,A -85,B 0,C 180,E1 -26088.515,E2 -26088.515} C_VEL
LIN {X 0,Y 141.723,Z 420.161,A -85,B 0,C 180,E1 -26091.442,E2 -26091.442} C_VEL
LIN {X 0,Y 142.451,Z 423.395,A -85,B 0,C 180,E1 -26097.169,E2 -26097.169} C_VEL
LIN {X 0,Y 142.524,Z 428.284,A -85,B 0,C 180,E1 -26102.824,E2 -26102.824} C_VEL
LIN {X 0,Y 142.279,Z 431.168,A -85,B 0,C 180,E1 -26105.667,E2 -26105.667} C_VEL
LIN {X 0,Y 141.425,Z 434.501,A -85,B 0,C 180,E1 -26108.571,E2 -26108.571} C_VEL
LIN {X 0,Y 139.631,Z 438.223,A -85,B 0,C 180,E1 -26111.612,E2 -26111.612} C_VEL
LIN {X 0,Y 135.824,Z 442.043,A -85,B 0,C 180,E1 -26114.087,E2 -26114.087} C_VEL
LIN {X 0,Y 132.444,Z 444.686,A -85,B 0,C 180,E1 -26115.846,E2 -26115.846} C_VEL
LIN {X 0,Y 125.519,Z 448.421,A -85,B 0,C 180,E1 -26118.544,E2 -26118.544} C_VEL
LIN {X 0,Y 118.735,Z 451.243,A -85,B 0,C 180,E1 -26121.656,E2 -26121.656} C_VEL
LIN {X 0,Y 115.688,Z 452.423,A -85,B 0,C 180,E1 -26124.039,E2 -26124.039} C_VEL
LIN {X 0,Y 112.073,Z 453.535,A -85,B 0,C 180,E1 -26128.598,E2 -26128.598} C_VEL
LIN {X 0,Y 109.267,Z 453.743,A -85,B 0,C 180,E1 -26133.256,E2 -26133.256} C_VEL
LIN {X 0,Y 107.127,Z 453.119,A -85,B 0,C 180,E1 -26138.064,E2 -26138.064} C_VEL
LIN {X 0,Y 105.746,Z 451.655,A -85,B 0,C 180,E1 -26143.017,E2 -26143.017} C_VEL
LIN {X 0,Y 105.054,Z 449.348,A -85,B 0,C 180,E1 -26148.005,E2 -26148.005} C_VEL
LIN {X 0,Y 105.066,Z 445.829,A -85,B 0,C 180,E1 -26153.381,E2 -26153.381} C_VEL
LIN {X 0,Y 105.647,Z 442.029,A -85,B 0,C 180,E1 -26157.841,E2 -26157.841} C_VEL
LIN {X 0,Y 106.809,Z 436.876,A -85,B 0,C 180,E1 -26162.569,E2 -26162.569} C_VEL
LIN {X 0,Y 107.861,Z 432.604,A -85,B 0,C 180,E1 -26165.802,E2 -26165.802} C_VEL
LIN {X 0,Y 109.853,Z 424.958,A -85,B 0,C 180,E1 -26170.369,E2 -26170.369} C_VEL
LIN {X 0,Y 111.486,Z 418.39,A -85,B 0,C 180,E1 -26173.516,E2 -26173.516} C_VEL
LIN {X 0,Y 113.207,Z 411.85,A -85,B 0,C 180,E1 -26176.076,E2 -26176.076} C_VEL
LIN {X 0,Y 113.023,Z 405.788,A -85,B 0,C 180,E1 -26178.336,E2 -26178.336} C_VEL
LIN {X 0,Y 112.238,Z 397.67,A -85,B 0,C 180,E1 -26180.989,E2 -26180.989} C_VEL
LIN {X 0,Y 111.049,Z 390.025,A -85,B 0,C 180,E1 -26183.18,E2 -26183.18} C_VEL
LIN {X 0,Y 108.264,Z 379.816,A -85,B 0,C 180,E1 -26185.924,E2 -26185.924} C_VEL
LIN {X 0,Y 108.878,Z 379.738,A -85,B 0,C 180,E1 -26189.995,E2 -26189.995} C_VEL
LIN {X 0,Y 108.332,Z 379.803,A -85,B 0,C 180,E1 -26197.45,E2 -26197.45} C_VEL
LIN {X 0,Y 108.194,Z 379.816,A -85,B 0,C 180,E1 -26203.021,E2 -26203.021} C_VEL
LIN {X 0,Y 107.898,Z 379.852,A -85,B 0,C 180,E1 -26209.001,E2 -26209.001} C_VEL
LIN {X 0,Y 107.847,Z 379.863,A -85,B 0,C 180,E1 -26214.181,E2 -26214.181} C_VEL
LIN {X 0,Y 107.789,Z 379.871,A -85,B 0,C 180,E1 -26222.054,E2 -26222.054} C_VEL
LIN {X 0,Y 107.774,Z 379.87,A -85,B 0,C 180,E1 -26228.514,E2 -26228.514} C_VEL
LIN {X 0,Y 107.776,Z 379.868,A -85,B 0,C 180,E1 -26235.825,E2 -26235.825} C_VEL
LIN {X 0,Y 107.773,Z 379.869,A -85,B 0,C 180,E1 -26241.485,E2 -26241.485} C_VEL
LIN {X 0,Y 107.799,Z 379.869,A -85,B 0,C 180,E1 -26248.568,E2 -26248.568} C_VEL
LIN {X 0,Y 107.921,Z 379.853,A -85,B 0,C 180,E1 -26257.004,E2 -26257.004} C_VEL
LIN {X 0,Y 108.041,Z 379.838,A -85,B 0,C 180,E1 -26264.922,E2 -26264.922} C_VEL
LIN {X 0,Y 108.304,Z 379.802,A -85,B 0,C 180,E1 -26268.778,E2 -26268.778} C_VEL
LIN {X 0,Y 108.452,Z 379.782,A -85,B 0,C 180,E1 -26276.288,E2 -26276.288} C_VEL
LIN {X 0,Y 108.937,Z 379.729,A -85,B 0,C 180,E1 -26280.004,E2 -26280.004} C_VEL
LIN {X 0,Y 108.328,Z 379.803,A -85,B 0,C 180,E1 -26287.459,E2 -26287.459} C_VEL
LIN {X 0,Y 108.194,Z 379.813,A -85,B 0,C 180,E1 -26293.027,E2 -26293.027} C_VEL
LIN {X 0,Y 107.9,Z 379.855,A -85,B 0,C 180,E1 -26299.01,E2 -26299.01} C_VEL
LIN {X 0,Y 107.851,Z 379.862,A -85,B 0,C 180,E1 -26304.189,E2 -26304.189} C_VEL
LIN {X 0,Y 107.783,Z 379.871,A -85,B 0,C 180,E1 -26312.051,E2 -26312.051} C_VEL
LIN {X 0,Y 107.725,Z 379.873,A -85,B 0,C 180,E1 -26318.483,E2 -26318.483} C_VEL
LIN {X 0,Y 108.228,Z 379.814,A -85,B 0,C 180,E1 -26326.931,E2 -26326.931} C_VEL
LIN {X 0,Y 108.714,Z 382.699,A -85,B 0,C 180,E1 -26332.912,E2 -26332.912} C_VEL
LIN {X 0,Y 108.7,Z 382.867,A -85,B 0,C 180,E1 -26333.242,E2 -26333.242} C_VEL
LIN {X 0,Y 109.91,Z 391.003,A -85,B 0,C 180,E1 -26334.79,E2 -26334.79} C_VEL
LIN {X 0,Y 110.501,Z 402.594,A -85,B 0,C 180,E1 -26337.34,E2 -26337.34} C_VEL
LIN {X 0,Y 110.672,Z 412.003,A -85,B 0,C 180,E1 -26340.019,E2 -26340.019} C_VEL
LIN {X 0,Y 110.525,Z 420.406,A -85,B 0,C 180,E1 -26342.908,E2 -26342.908} C_VEL
LIN {X 0,Y 110.201,Z 427.949,A -85,B 0,C 180,E1 -26346.016,E2 -26346.016} C_VEL
LIN {X 0,Y 109.72,Z 432.987,A -85,B 0,C 180,E1 -26348.394,E2 -26348.394} C_VEL
LIN {X 0,Y 108.097,Z 439.441,A -85,B 0,C 180,E1 -26352.017,E2 -26352.017} C_VEL
LIN {X 0,Y 106.89,Z 444.822,A -85,B 0,C 180,E1 -26355.731,E2 -26355.731} C_VEL
LIN {X 0,Y 105.957,Z 450.256,A -85,B 0,C 180,E1 -26360.46,E2 -26360.46} C_VEL
LIN {X 0,Y 105.679,Z 455.289,A -85,B 0,C 180,E1 -26366.192,E2 -26366.192} C_VEL
LIN {X 0,Y 105.781,Z 457.806,A -85,B 0,C 180,E1 -26370.005,E2 -26370.005} C_VEL
LIN {X 0,Y 105.489,Z 459.692,A -85,B 0,C 180,E1 -26373.825,E2 -26373.825} C_VEL
LIN {X 0,Y 105.547,Z 461.089,A -85,B 0,C 180,E1 -26377.658,E2 -26377.658} C_VEL
LIN {X 0,Y 106.053,Z 461.911,A -85,B 0,C 180,E1 -26381.472,E2 -26381.472} C_VEL
LIN {X 0,Y 107.024,Z 462.293,A -85,B 0,C 180,E1 -26385.233,E2 -26385.233} C_VEL
LIN {X 0,Y 108.422,Z 462.27,A -85,B 0,C 180,E1 -26388.916,E2 -26388.916} C_VEL
LIN {X 0,Y 110.261,Z 461.81,A -85,B 0,C 180,E1 -26392.49,E2 -26392.49} C_VEL
LIN {X 0,Y 112.627,Z 460.79,A -85,B 0,C 180,E1 -26395.905,E2 -26395.905} C_VEL
LIN {X 0,Y 115.452,Z 459.338,A -85,B 0,C 180,E1 -26399.148,E2 -26399.148} C_VEL
LIN {X 0,Y 120.44,Z 456.279,A -85,B 0,C 180,E1 -26403.671,E2 -26403.671} C_VEL
LIN {X 0,Y 125.923,Z 452.059,A -85,B 0,C 180,E1 -26407.879,E2 -26407.879} C_VEL
LIN {X 0,Y 129.173,Z 448.524,A -85,B 0,C 180,E1 -26410.765,E2 -26410.765} C_VEL
LIN {X 0,Y 132.876,Z 443.463,A -85,B 0,C 180,E1 -26414.497,E2 -26414.497} C_VEL
LIN {X 0,Y 135.41,Z 439.035,A -85,B 0,C 180,E1 -26417.564,E2 -26417.564} C_VEL
LIN {X 0,Y 135.892,Z 435.646,A -85,B 0,C 180,E1 -26420.88,E2 -26420.88} C_VEL
LIN {X 0,Y 136.039,Z 431.262,A -85,B 0,C 180,E1 -26425.756,E2 -26425.756} C_VEL
LIN {X 0,Y 136.03,Z 429.013,A -85,B 0,C 180,E1 -26428.889,E2 -26428.889} C_VEL
LIN {X 0,Y 135.941,Z 427.067,A -85,B 0,C 180,E1 -26432.268,E2 -26432.268} C_VEL
LIN {X 0,Y 135.773,Z 425.704,A -85,B 0,C 180,E1 -26435.534,E2 -26435.534} C_VEL
LIN {X 0,Y 135.743,Z 424.833,A -85,B 0,C 180,E1 -26438.748,E2 -26438.748} C_VEL
LIN {X 0,Y 135.863,Z 424.326,A -85,B 0,C 180,E1 -26441.915,E2 -26441.915} C_VEL
LIN {X 0,Y 136.443,Z 424.635,A -85,B 0,C 180,E1 -26448.16,E2 -26448.16} C_VEL
LIN {X 0,Y 136.908,Z 425.358,A -85,B 0,C 180,E1 -26451.138,E2 -26451.138} C_VEL
LIN {X 0,Y 137.194,Z 428.316,A -85,B 0,C 180,E1 -26457.061,E2 -26457.061} C_VEL
LIN {X 0,Y 136.914,Z 431.697,A -85,B 0,C 180,E1 -26461.468,E2 -26461.468} C_VEL
LIN {X 0,Y 136.525,Z 434.253,A -85,B 0,C 180,E1 -26464.426,E2 -26464.426} C_VEL
LIN {X 0,Y 135.431,Z 437.234,A -85,B 0,C 180,E1 -26467.411,E2 -26467.411} C_VEL
LIN {X 0,Y 134.008,Z 439.873,A -85,B 0,C 180,E1 -26469.811,E2 -26469.811} C_VEL
LIN {X 0,Y 132.939,Z 441,A -85,B 0,C 180,E1 -26470.66,E2 -26470.66} C_VEL
LIN {X 0,Y 126.978,Z 445.842,A -85,B 0,C 180,E1 -26474.383,E2 -26474.383} C_VEL
LIN {X 0,Y 121.825,Z 449.279,A -85,B 0,C 180,E1 -26478.204,E2 -26478.204} C_VEL
LIN {X 0,Y 118.922,Z 450.935,A -85,B 0,C 180,E1 -26480.764,E2 -26480.764} C_VEL
LIN {X 0,Y 115.688,Z 452.423,A -85,B 0,C 180,E1 -26484.039,E2 -26484.039} C_VEL
LIN {X 0,Y 112.825,Z 453.347,A -85,B 0,C 180,E1 -26486.583,E2 -26486.583} C_VEL
LIN {X 0,Y 106.934,Z 453.913,A -85,B 0,C 180,E1 -26490.725,E2 -26490.725} C_VEL
LIN {X 0,Y 102.513,Z 453.738,A -85,B 0,C 180,E1 -26494.35,E2 -26494.35} C_VEL
LIN {X 0,Y 100.203,Z 453.175,A -85,B 0,C 180,E1 -26497.425,E2 -26497.425} C_VEL
LIN {X 0,Y 99.749,Z 452.853,A -85,B 0,C 180,E1 -26498.522,E2 -26498.522} C_VEL
LIN {X 0,Y 98.143,Z 450.284,A -85,B 0,C 180,E1 -26505.727,E2 -26505.727} C_VEL
LIN {X 0,Y 97.921,Z 446.572,A -85,B 0,C 180,E1 -26512.131,E2 -26512.131} C_VEL
LIN {X 0,Y 98.687,Z 441.19,A -85,B 0,C 180,E1 -26518.705,E2 -26518.705} C_VEL
LIN {X 0,Y 100.052,Z 435.534,A -85,B 0,C 180,E1 -26523.953,E2 -26523.953} C_VEL
LIN {X 0,Y 101.769,Z 428.949,A -85,B 0,C 180,E1 -26528.737,E2 -26528.737} C_VEL
LIN {X 0,Y 104.123,Z 420.199,A -85,B 0,C 180,E1 -26533.56,E2 -26533.56} C_VEL
LIN {X 0,Y 106.367,Z 411.803,A -85,B 0,C 180,E1 -26537.11,E2 -26537.11} C_VEL
LIN {X 0,Y 105.992,Z 404.454,A -85,B 0,C 180,E1 -26539.971,E2 -26539.971} C_VEL
LIN {X 0,Y 105.182,Z 396.05,A -85,B 0,C 180,E1 -26542.798,E2 -26542.798} C_VEL
LIN {X 0,Y 103.593,Z 388.504,A -85,B 0,C 180,E1 -26545.13,E2 -26545.13} C_VEL
LIN {X 0,Y 101.398,Z 380.67,A -85,B 0,C 180,E1 -26547.512,E2 -26547.512} C_VEL
LIN {X 0,Y 101.797,Z 380.62,A -85,B 0,C 180,E1 -26549.995,E2 -26549.995} C_VEL
LIN {X 0,Y 101.271,Z 380.683,A -85,B 0,C 180,E1 -26557.973,E2 -26557.973} C_VEL
LIN {X 0,Y 101.12,Z 380.698,A -85,B 0,C 180,E1 -26563.358,E2 -26563.358} C_VEL
LIN {X 0,Y 100.808,Z 380.734,A -85,B 0,C 180,E1 -26570.395,E2 -26570.395} C_VEL
LIN {X 0,Y 100.764,Z 380.746,A -85,B 0,C 180,E1 -26574.956,E2 -26574.956} C_VEL
LIN {X 0,Y 100.7,Z 380.754,A -85,B 0,C 180,E1 -26583.131,E2 -26583.131} C_VEL
LIN {X 0,Y 100.716,Z 380.752,A -85,B 0,C 180,E1 -26589.87,E2 -26589.87} C_VEL
LIN {X 0,Y 100.741,Z 380.744,A -85,B 0,C 180,E1 -26595.769,E2 -26595.769} C_VEL
LIN {X 0,Y 100.714,Z 380.749,A -85,B 0,C 180,E1 -26601.1,E2 -26601.1} C_VEL
LIN {X 0,Y 100.699,Z 380.755,A -85,B 0,C 180,E1 -26606.867,E2 -26606.867} C_VEL
LIN {X 0,Y 100.775,Z 380.744,A -85,B 0,C 180,E1 -26615.269,E2 -26615.269} C_VEL
LIN {X 0,Y 100.827,Z 380.73,A -85,B 0,C 180,E1 -26619.608,E2 -26619.608} C_VEL
LIN {X 0,Y 101.2,Z 380.685,A -85,B 0,C 180,E1 -26627.979,E2 -26627.979} C_VEL
LIN {X 0,Y 101.27,Z 380.684,A -85,B 0,C 180,E1 -26632.026,E2 -26632.026} C_VEL
LIN {X 0,Y 101.862,Z 380.61,A -85,B 0,C 180,E1 -26640.004,E2 -26640.004} C_VEL
LIN {X 0,Y 101.268,Z 380.684,A -85,B 0,C 180,E1 -26647.982,E2 -26647.982} C_VEL
LIN {X 0,Y 101.12,Z 380.694,A -85,B 0,C 180,E1 -26653.364,E2 -26653.364} C_VEL
LIN {X 0,Y 100.811,Z 380.733,A -85,B 0,C 180,E1 -26660.404,E2 -26660.404} C_VEL
LIN {X 0,Y 100.769,Z 380.745,A -85,B 0,C 180,E1 -26664.964,E2 -26664.964} C_VEL
LIN {X 0,Y 100.691,Z 380.756,A -85,B 0,C 180,E1 -26673.126,E2 -26673.126} C_VEL
LIN {X 0,Y 100.695,Z 380.753,A -85,B 0,C 180,E1 -26679.857,E2 -26679.857} C_VEL
LIN {X 0,Y 101.235,Z 380.797,A -85,B 0,C 180,E1 -26687.667,E2 -26687.667} C_VEL
LIN {X 0,Y 101.544,Z 382.544,A -85,B 0,C 180,E1 -26691.479,E2 -26691.479} C_VEL
LIN {X 0,Y 103.175,Z 390.656,A -85,B 0,C 180,E1 -26693.282,E2 -26693.282} C_VEL
LIN {X 0,Y 103.709,Z 401.943,A -85,B 0,C 180,E1 -26695.912,E2 -26695.912} C_VEL
LIN {X 0,Y 103.781,Z 411.888,A -85,B 0,C 180,E1 -26698.918,E2 -26698.918} C_VEL
LIN {X 0,Y 103.549,Z 421.142,A -85,B 0,C 180,E1 -26702.358,E2 -26702.358} C_VEL
LIN {X 0,Y 103.195,Z 427.869,A -85,B 0,C 180,E1 -26705.352,E2 -26705.352} C_VEL
LIN {X 0,Y 103.046,Z 431.064,A -85,B 0,C 180,E1 -26706.916,E2 -26706.916} C_VEL
LIN {X 0,Y 100.987,Z 439.267,A -85,B 0,C 180,E1 -26711.755,E2 -26711.755} C_VEL
LIN {X 0,Y 99.785,Z 444.61,A -85,B 0,C 180,E1 -26715.734,E2 -26715.734} C_VEL
LIN {X 0,Y 98.976,Z 449.064,A -85,B 0,C 180,E1 -26719.78,E2 -26719.78} C_VEL
LIN {X 0,Y 98.602,Z 452.757,A -85,B 0,C 180,E1 -26723.868,E2 -26723.868} C_VEL
LIN {X 0,Y 98.722,Z 456.934,A -85,B 0,C 180,E1 -26730.005,E2 -26730.005} C_VEL
LIN {X 0,Y 98.428,Z 458.969,A -85,B 0,C 180,E1 -26734.1,E2 -26734.1} C_VEL
LIN {X 0,Y 98.543,Z 460.403,A -85,B 0,C 180,E1 -26738.206,E2 -26738.206} C_VEL
LIN {X 0,Y 99.125,Z 461.348,A -85,B 0,C 180,E1 -26742.286,E2 -26742.286} C_VEL
LIN {X 0,Y 100.171,Z 461.878,A -85,B 0,C 180,E1 -26746.304,E2 -26746.304} C_VEL
LIN {X 0,Y 101.73,Z 462,A -85,B 0,C 180,E1 -26750.213,E2 -26750.213} C_VEL
LIN {X 0,Y 103.718,Z 461.57,A -85,B 0,C 180,E1 -26753.994,E2 -26753.994} C_VEL
LIN {X 0,Y 106.292,Z 460.697,A -85,B 0,C 180,E1 -26757.576,E2 -26757.576} C_VEL
LIN {X 0,Y 109.312,Z 459.409,A -85,B 0,C 180,E1 -26760.959,E2 -26760.959} C_VEL
LIN {X 0,Y 114.603,Z 456.521,A -85,B 0,C 180,E1 -26765.638,E2 -26765.638} C_VEL
LIN {X 0,Y 118.5,Z 453.985,A -85,B 0,C 180,E1 -26768.521,E2 -26768.521} C_VEL
LIN {X 0,Y 122.508,Z 450.604,A -85,B 0,C 180,E1 -26771.77,E2 -26771.77} C_VEL
LIN {X 0,Y 126.99,Z 445.478,A -85,B 0,C 180,E1 -26776.015,E2 -26776.015} C_VEL
LIN {X 0,Y 129.259,Z 442.271,A -85,B 0,C 180,E1 -26778.469,E2 -26778.469} C_VEL
LIN {X 0,Y 129.713,Z 441.258,A -85,B 0,C 180,E1 -26779.442,E2 -26779.442} C_VEL
LIN {X 0,Y 130.312,Z 437.335,A -85,B 0,C 180,E1 -26784.002,E2 -26784.002} C_VEL
LIN {X 0,Y 130.619,Z 434.834,A -85,B 0,C 180,E1 -26787.446,E2 -26787.446} C_VEL
LIN {X 0,Y 130.754,Z 432.637,A -85,B 0,C 180,E1 -26791.066,E2 -26791.066} C_VEL
LIN {X 0,Y 130.741,Z 430.591,A -85,B 0,C 180,E1 -26796.049,E2 -26796.049} C_VEL
LIN {X 0,Y 130.84,Z 429.518,A -85,B 0,C 180,E1 -26801.196,E2 -26801.196} C_VEL
LIN {X 0,Y 131.068,Z 429.392,A -85,B 0,C 180,E1 -26804.848,E2 -26804.848} C_VEL
LIN {X 0,Y 131.308,Z 429.575,A -85,B 0,C 180,E1 -26807.635,E2 -26807.635} C_VEL
LIN {X 0,Y 131.705,Z 430.159,A -85,B 0,C 180,E1 -26810.785,E2 -26810.785} C_VEL
LIN {X 0,Y 131.686,Z 431.462,A -85,B 0,C 180,E1 -26813.87,E2 -26813.87} C_VEL
LIN {X 0,Y 131.668,Z 432.924,A -85,B 0,C 180,E1 -26816.937,E2 -26816.937} C_VEL
LIN {X 0,Y 131.05,Z 436.087,A -85,B 0,C 180,E1 -26821.533,E2 -26821.533} C_VEL
LIN {X 0,Y 130.183,Z 438.489,A -85,B 0,C 180,E1 -26824.642,E2 -26824.642} C_VEL
LIN {X 0,Y 128.567,Z 441.37,A -85,B 0,C 180,E1 -26827.767,E2 -26827.767} C_VEL
LIN {X 0,Y 127.898,Z 442.071,A -85,B 0,C 180,E1 -26828.442,E2 -26828.442} C_VEL
LIN {X 0,Y 122.134,Z 446.423,A -85,B 0,C 180,E1 -26831.958,E2 -26831.958} C_VEL
LIN {X 0,Y 116.802,Z 449.69,A -85,B 0,C 180,E1 -26835.68,E2 -26835.68} C_VEL
LIN {X 0,Y 112.024,Z 452.023,A -85,B 0,C 180,E1 -26839.76,E2 -26839.76} C_VEL
LIN {X 0,Y 107.843,Z 453.465,A -85,B 0,C 180,E1 -26844.155,E2 -26844.155} C_VEL
LIN {X 0,Y 104.366,Z 454.056,A -85,B 0,C 180,E1 -26848.896,E2 -26848.896} C_VEL
LIN {X 0,Y 101.6,Z 453.811,A -85,B 0,C 180,E1 -26853.885,E2 -26853.885} C_VEL
LIN {X 0,Y 99.749,Z 452.853,A -85,B 0,C 180,E1 -26858.522,E2 -26858.522} C_VEL
LIN {X 0,Y 98.18,Z 451.933,A -85,B 0,C 180,E1 -26861.77,E2 -26861.77} C_VEL
LIN {X 0,Y 96,Z 450.562,A -85,B 0,C 180,E1 -26864.933,E2 -26864.933} C_VEL
LIN {X 0,Y 91.911,Z 446.857,A -85,B 0,C 180,E1 -26871.397,E2 -26871.397} C_VEL
LIN {X 0,Y 91.085,Z 444.462,A -85,B 0,C 180,E1 -26874.793,E2 -26874.793} C_VEL
LIN {X 0,Y 91.136,Z 443.621,A -85,B 0,C 180,E1 -26875.932,E2 -26875.932} C_VEL
LIN {X 0,Y 92.197,Z 438.49,A -85,B 0,C 180,E1 -26881.614,E2 -26881.614} C_VEL
LIN {X 0,Y 93.811,Z 432.268,A -85,B 0,C 180,E1 -26886.955,E2 -26886.955} C_VEL
LIN {X 0,Y 95.612,Z 425.854,A -85,B 0,C 180,E1 -26891.32,E2 -26891.32} C_VEL
LIN {X 0,Y 97.402,Z 419.48,A -85,B 0,C 180,E1 -26894.832,E2 -26894.832} C_VEL
LIN {X 0,Y 99.229,Z 413.059,A -85,B 0,C 180,E1 -26897.727,E2 -26897.727} C_VEL
LIN {X 0,Y 99.402,Z 409.442,A -85,B 0,C 180,E1 -26899.299,E2 -26899.299} C_VEL
LIN {X 0,Y 98.646,Z 398.973,A -85,B 0,C 180,E1 -26903.347,E2 -26903.347} C_VEL
LIN {X 0,Y 97.37,Z 391.791,A -85,B 0,C 180,E1 -26905.856,E2 -26905.856} C_VEL
LIN {X 0,Y 94.566,Z 381.521,A -85,B 0,C 180,E1 -26909.196,E2 -26909.196} C_VEL
LIN {X 0,Y 94.721,Z 381.501,A -85,B 0,C 180,E1 -26909.995,E2 -26909.995} C_VEL
LIN {X 0,Y 94.203,Z 381.562,A -85,B 0,C 180,E1 -26918.576,E2 -26918.576} C_VEL
LIN {X 0,Y 94.038,Z 381.581,A -85,B 0,C 180,E1 -26923.716,E2 -26923.716} C_VEL
LIN {X 0,Y 93.684,Z 381.625,A -85,B 0,C 180,E1 -26932.024,E2 -26932.024} C_VEL
LIN {X 0,Y 93.613,Z 381.633,A -85,B 0,C 180,E1 -26936.766,E2 -26936.766} C_VEL
LIN {X 0,Y 93.612,Z 381.635,A -85,B 0,C 180,E1 -26944.335,E2 -26944.335} C_VEL
LIN {X 0,Y 93.637,Z 381.632,A -85,B 0,C 180,E1 -26952.485,E2 -26952.485} C_VEL
LIN {X 0,Y 93.635,Z 381.634,A -85,B 0,C 180,E1 -26958.631,E2 -26958.631} C_VEL
LIN {X 0,Y 93.611,Z 381.636,A -85,B 0,C 180,E1 -26965.663,E2 -26965.663} C_VEL
LIN {X 0,Y 93.658,Z 381.63,A -85,B 0,C 180,E1 -26974.206,E2 -26974.206} C_VEL
LIN {X 0,Y 93.695,Z 381.622,A -85,B 0,C 180,E1 -26977.978,E2 -26977.978} C_VEL
LIN {X 0,Y 94.1,Z 381.57,A -85,B 0,C 180,E1 -26987.057,E2 -26987.057} C_VEL
LIN {X 0,Y 94.204,Z 381.563,A -85,B 0,C 180,E1 -26991.423,E2 -26991.423} C_VEL
LIN {X 0,Y 94.788,Z 381.491,A -85,B 0,C 180,E1 -27000.004,E2 -27000.004} C_VEL
LIN {X 0,Y 94.2,Z 381.563,A -85,B 0,C 180,E1 -27008.586,E2 -27008.586} C_VEL
LIN {X 0,Y 94.038,Z 381.577,A -85,B 0,C 180,E1 -27013.723,E2 -27013.723} C_VEL
LIN {X 0,Y 93.688,Z 381.622,A -85,B 0,C 180,E1 -27022.033,E2 -27022.033} C_VEL
LIN {X 0,Y 93.615,Z 381.635,A -85,B 0,C 180,E1 -27026.776,E2 -27026.776} C_VEL
LIN {X 0,Y 93.594,Z 381.639,A -85,B 0,C 180,E1 -27034.321,E2 -27034.321} C_VEL
LIN {X 0,Y 93.729,Z 381.622,A -85,B 0,C 180,E1 -27042.447,E2 -27042.447} C_VEL
LIN {X 0,Y 94.205,Z 381.682,A -85,B 0,C 180,E1 -27048.253,E2 -27048.253} C_VEL
LIN {X 0,Y 94.327,Z 382.429,A -85,B 0,C 180,E1 -27049.488,E2 -27049.488} C_VEL
LIN {X 0,Y 96.369,Z 390.289,A -85,B 0,C 180,E1 -27051.527,E2 -27051.527} C_VEL
LIN {X 0,Y 96.886,Z 399.48,A -85,B 0,C 180,E1 -27053.831,E2 -27053.831} C_VEL
LIN {X 0,Y 96.952,Z 410.064,A -85,B 0,C 180,E1 -27057.073,E2 -27057.073} C_VEL
LIN {X 0,Y 96.64,Z 419.595,A -85,B 0,C 180,E1 -27060.779,E2 -27060.779} C_VEL
LIN {X 0,Y 96.29,Z 426.585,A -85,B 0,C 180,E1 -27064.035,E2 -27064.035} C_VEL
LIN {X 0,Y 96.028,Z 430.841,A -85,B 0,C 180,E1 -27066.27,E2 -27066.27} C_VEL
LIN {X 0,Y 93.907,Z 439.013,A -85,B 0,C 180,E1 -27071.46,E2 -27071.46} C_VEL
LIN {X 0,Y 92.668,Z 444.336,A -85,B 0,C 180,E1 -27075.736,E2 -27075.736} C_VEL
LIN {X 0,Y 91.738,Z 449.709,A -85,B 0,C 180,E1 -27081.192,E2 -27081.192} C_VEL
LIN {X 0,Y 91.589,Z 454.588,A -85,B 0,C 180,E1 -27087.666,E2 -27087.666} C_VEL
LIN {X 0,Y 91.666,Z 456.06,A -85,B 0,C 180,E1 -27090.006,E2 -27090.006} C_VEL
LIN {X 0,Y 91.397,Z 458.153,A -85,B 0,C 180,E1 -27094.416,E2 -27094.416} C_VEL
LIN {X 0,Y 91.56,Z 459.684,A -85,B 0,C 180,E1 -27098.836,E2 -27098.836} C_VEL
LIN {X 0,Y 92.195,Z 460.773,A -85,B 0,C 180,E1 -27103.225,E2 -27103.225} C_VEL
LIN {X 0,Y 93.369,Z 461.458,A -85,B 0,C 180,E1 -27107.528,E2 -27107.528} C_VEL
LIN {X 0,Y 95.083,Z 461.631,A -85,B 0,C 180,E1 -27111.695,E2 -27111.695} C_VEL
LIN {X 0,Y 97.259,Z 461.312,A -85,B 0,C 180,E1 -27115.7,E2 -27115.7} C_VEL
LIN {X 0,Y 100.061,Z 460.603,A -85,B 0,C 180,E1 -27119.455,E2 -27119.455} C_VEL
LIN {X 0,Y 103.297,Z 459.478,A -85,B 0,C 180,E1 -27122.982,E2 -27122.982} C_VEL
LIN {X 0,Y 108.918,Z 456.787,A -85,B 0,C 180,E1 -27127.812,E2 -27127.812} C_VEL
LIN {X 0,Y 113.036,Z 454.441,A -85,B 0,C 180,E1 -27130.761,E2 -27130.761} C_VEL
LIN {X 0,Y 116.867,Z 451.489,A -85,B 0,C 180,E1 -27133.806,E2 -27133.806} C_VEL
LIN {X 0,Y 122.032,Z 446.368,A -85,B 0,C 180,E1 -27138.483,E2 -27138.483} C_VEL
LIN {X 0,Y 123.586,Z 444.283,A -85,B 0,C 180,E1 -27140.317,E2 -27140.317} C_VEL
LIN {X 0,Y 124.654,Z 440.397,A -85,B 0,C 180,E1 -27145.677,E2 -27145.677} C_VEL
LIN {X 0,Y 125.095,Z 437.944,A -85,B 0,C 180,E1 -27149.623,E2 -27149.623} C_VEL
LIN {X 0,Y 125.233,Z 436.064,A -85,B 0,C 180,E1 -27153.893,E2 -27153.893} C_VEL
LIN {X 0,Y 125.413,Z 435.104,A -85,B 0,C 180,E1 -27156.901,E2 -27156.901} C_VEL
LIN {X 0,Y 125.584,Z 434.25,A -85,B 0,C 180,E1 -27162.069,E2 -27162.069} C_VEL
LIN {X 0,Y 125.926,Z 434.227,A -85,B 0,C 180,E1 -27167.097,E2 -27167.097} C_VEL
LIN {X 0,Y 126.207,Z 434.664,A -85,B 0,C 180,E1 -27170.38,E2 -27170.38} C_VEL
LIN {X 0,Y 126.084,Z 435.772,A -85,B 0,C 180,E1 -27173.596,E2 -27173.596} C_VEL
LIN {X 0,Y 125.884,Z 437.21,A -85,B 0,C 180,E1 -27176.796,E2 -27176.796} C_VEL
LIN {X 0,Y 124.84,Z 440.043,A -85,B 0,C 180,E1 -27181.61,E2 -27181.61} C_VEL
LIN {X 0,Y 123.475,Z 442.396,A -85,B 0,C 180,E1 -27184.894,E2 -27184.894} C_VEL
LIN {X 0,Y 122.257,Z 443.834,A -85,B 0,C 180,E1 -27186.599,E2 -27186.599} C_VEL
LIN {X 0,Y 114.619,Z 448.837,A -85,B 0,C 180,E1 -27191.148,E2 -27191.148} C_VEL
LIN {X 0,Y 109.199,Z 451.537,A -85,B 0,C 180,E1 -27195.102,E2 -27195.102} C_VEL
LIN {X 0,Y 104.006,Z 453.419,A -85,B 0,C 180,E1 -27199.743,E2 -27199.743} C_VEL
LIN {X 0,Y 99.386,Z 454.353,A -85,B 0,C 180,E1 -27205.101,E2 -27205.101} C_VEL
LIN {X 0,Y 95.7,Z 454.25,A -85,B 0,C 180,E1 -27210.93,E2 -27210.93} C_VEL
LIN {X 0,Y 92.959,Z 453.085,A -85,B 0,C 180,E1 -27217.21,E2 -27217.21} C_VEL
LIN {X 0,Y 91.321,Z 450.814,A -85,B 0,C 180,E1 -27223.832,E2 -27223.832} C_VEL
LIN {X 0,Y 90.821,Z 446.562,A -85,B 0,C 180,E1 -27231.745,E2 -27231.745} C_VEL
LIN {X 0,Y 91.136,Z 443.621,A -85,B 0,C 180,E1 -27235.932,E2 -27235.932} C_VEL
LIN {X 0,Y 90.977,Z 440.916,A -85,B 0,C 180,E1 -27239.237,E2 -27239.237} C_VEL
LIN {X 0,Y 90.048,Z 437.848,A -85,B 0,C 180,E1 -27242.418,E2 -27242.418} C_VEL
LIN {X 0,Y 88.114,Z 429.61,A -85,B 0,C 180,E1 -27249.557,E2 -27249.557} C_VEL
LIN {X 0,Y 88.756,Z 425.518,A -85,B 0,C 180,E1 -27252.38,E2 -27252.38} C_VEL
LIN {X 0,Y 90.892,Z 418.194,A -85,B 0,C 180,E1 -27256.581,E2 -27256.581} C_VEL
LIN {X 0,Y 92.467,Z 412.907,A -85,B 0,C 180,E1 -27259.041,E2 -27259.041} C_VEL
LIN {X 0,Y 92.301,Z 405.857,A -85,B 0,C 180,E1 -27262.234,E2 -27262.234} C_VEL
LIN {X 0,Y 91.661,Z 398.091,A -85,B 0,C 180,E1 -27265.326,E2 -27265.326} C_VEL
LIN {X 0,Y 89.885,Z 390.216,A -85,B 0,C 180,E1 -27268.314,E2 -27268.314} C_VEL
LIN {X 0,Y 87.863,Z 383.75,A -85,B 0,C 180,E1 -27270.71,E2 -27270.71} C_VEL
LIN {X 0,Y 87.495,Z 382.401,A -85,B 0,C 180,E1 -27271.145,E2 -27271.145} C_VEL
LIN {X 0,Y 87.109,Z 382.445,A -85,B 0,C 180,E1 -27279.28,E2 -27279.28} C_VEL
LIN {X 0,Y 86.941,Z 382.466,A -85,B 0,C 180,E1 -27284.083,E2 -27284.083} C_VEL
LIN {X 0,Y 86.577,Z 382.513,A -85,B 0,C 180,E1 -27293.94,E2 -27293.94} C_VEL
LIN {X 0,Y 86.471,Z 382.52,A -85,B 0,C 180,E1 -27299.18,E2 -27299.18} C_VEL
LIN {X 0,Y 86.54,Z 382.511,A -85,B 0,C 180,E1 -27305.706,E2 -27305.706} C_VEL
LIN {X 0,Y 86.562,Z 382.511,A -85,B 0,C 180,E1 -27313.061,E2 -27313.061} C_VEL
LIN {X 0,Y 86.557,Z 382.515,A -85,B 0,C 180,E1 -27319.498,E2 -27319.498} C_VEL
LIN {X 0,Y 86.561,Z 382.513,A -85,B 0,C 180,E1 -27325.372,E2 -27325.372} C_VEL
LIN {X 0,Y 86.574,Z 382.51,A -85,B 0,C 180,E1 -27333.234,E2 -27333.234} C_VEL
LIN {X 0,Y 86.664,Z 382.498,A -85,B 0,C 180,E1 -27341.077,E2 -27341.077} C_VEL
LIN {X 0,Y 86.959,Z 382.462,A -85,B 0,C 180,E1 -27345.973,E2 -27345.973} C_VEL
LIN {X 0,Y 87.112,Z 382.446,A -85,B 0,C 180,E1 -27350.719,E2 -27350.719} C_VEL
LIN {X 0,Y 87.716,Z 382.372,A -85,B 0,C 180,E1 -27360.005,E2 -27360.005} C_VEL
LIN {X 0,Y 87.107,Z 382.447,A -85,B 0,C 180,E1 -27369.291,E2 -27369.291} C_VEL
LIN {X 0,Y 86.943,Z 382.462,A -85,B 0,C 180,E1 -27374.093,E2 -27374.093} C_VEL
LIN {X 0,Y 86.581,Z 382.512,A -85,B 0,C 180,E1 -27383.95,E2 -27383.95} C_VEL
LIN {X 0,Y 86.47,Z 382.519,A -85,B 0,C 180,E1 -27389.192,E2 -27389.192} C_VEL
LIN {X 0,Y 86.52,Z 382.517,A -85,B 0,C 180,E1 -27395.69,E2 -27395.69} C_VEL
LIN {X 0,Y 86.699,Z 382.496,A -85,B 0,C 180,E1 -27403.16,E2 -27403.16} C_VEL
LIN {X 0,Y 87.025,Z 382.517,A -85,B 0,C 180,E1 -27407.19,E2 -27407.19} C_VEL
LIN {X 0,Y 89.575,Z 390.239,A -85,B 0,C 180,E1 -27409.596,E2 -27409.596} C_VEL
LIN {X 0,Y 90.132,Z 396.204,A -85,B 0,C 180,E1 -27411.243,E2 -27411.243} C_VEL
LIN {X 0,Y 90.179,Z 406.037,A -85,B 0,C 180,E1 -27414.259,E2 -27414.259} C_VEL
LIN {X 0,Y 89.987,Z 415.038,A -85,B 0,C 180,E1 -27417.676,E2 -27417.676} C_VEL
LIN {X 0,Y 89.44,Z 425.299,A -85,B 0,C 180,E1 -27422.514,E2 -27422.514} C_VEL
LIN {X 0,Y 89.017,Z 430.614,A -85,B 0,C 180,E1 -27425.519,E2 -27425.519} C_VEL
LIN {X 0,Y 86.81,Z 438.754,A -85,B 0,C 180,E1 -27431.112,E2 -27431.112} C_VEL
LIN {X 0,Y 85.56,Z 444.064,A -85,B 0,C 180,E1 -27435.74,E2 -27435.74} C_VEL
LIN {X 0,Y 84.762,Z 448.483,A -85,B 0,C 180,E1 -27440.461,E2 -27440.461} C_VEL
LIN {X 0,Y 84.528,Z 453.475,A -85,B 0,C 180,E1 -27447.385,E2 -27447.385} C_VEL
LIN {X 0,Y 84.607,Z 455.066,A -85,B 0,C 180,E1 -27450.006,E2 -27450.006} C_VEL
LIN {X 0,Y 84.382,Z 457.248,A -85,B 0,C 180,E1 -27454.784,E2 -27454.784} C_VEL
LIN {X 0,Y 84.575,Z 458.938,A -85,B 0,C 180,E1 -27459.573,E2 -27459.573} C_VEL
LIN {X 0,Y 85.305,Z 460.191,A -85,B 0,C 180,E1 -27464.316,E2 -27464.316} C_VEL
LIN {X 0,Y 86.623,Z 460.968,A -85,B 0,C 180,E1 -27468.943,E2 -27468.943} C_VEL
LIN {X 0,Y 90.9,Z 461.057,A -85,B 0,C 180,E1 -27477.645,E2 -27477.645} C_VEL
LIN {X 0,Y 93.931,Z 460.521,A -85,B 0,C 180,E1 -27481.59,E2 -27481.59} C_VEL
LIN {X 0,Y 97.428,Z 459.476,A -85,B 0,C 180,E1 -27485.252,E2 -27485.252} C_VEL
LIN {X 0,Y 101.309,Z 457.918,A -85,B 0,C 180,E1 -27488.64,E2 -27488.64} C_VEL
LIN {X 0,Y 107.739,Z 454.763,A -85,B 0,C 180,E1 -27493.237,E2 -27493.237} C_VEL
LIN {X 0,Y 111.349,Z 452.303,A -85,B 0,C 180,E1 -27496.025,E2 -27496.025} C_VEL
LIN {X 0,Y 115.441,Z 448.913,A -85,B 0,C 180,E1 -27499.558,E2 -27499.558} C_VEL
LIN {X 0,Y 117.202,Z 447.193,A -85,B 0,C 180,E1 -27501.225,E2 -27501.225} C_VEL
LIN {X 0,Y 117.983,Z 445.705,A -85,B 0,C 180,E1 -27503.435,E2 -27503.435} C_VEL
LIN {X 0,Y 118.884,Z 442.989,A -85,B 0,C 180,E1 -27507.853,E2 -27507.853} C_VEL
LIN {X 0,Y 119.345,Z 441.063,A -85,B 0,C 180,E1 -27512.054,E2 -27512.054} C_VEL
LIN {X 0,Y 119.638,Z 439.84,A -85,B 0,C 180,E1 -27515.716,E2 -27515.716} C_VEL
LIN {X 0,Y 119.87,Z 438.966,A -85,B 0,C 180,E1 -27519.743,E2 -27519.743} C_VEL
LIN {X 0,Y 120.046,Z 438.616,A -85,B 0,C 180,E1 -27522.976,E2 -27522.976} C_VEL
LIN {X 0,Y 120.258,Z 438.577,A -85,B 0,C 180,E1 -27526.478,E2 -27526.478} C_VEL
LIN {X 0,Y 120.481,Z 438.842,A -85,B 0,C 180,E1 -27529.918,E2 -27529.918} C_VEL
LIN {X 0,Y 120.134,Z 440.024,A -85,B 0,C 180,E1 -27534.037,E2 -27534.037} C_VEL
LIN {X 0,Y 119.608,Z 441.456,A -85,B 0,C 180,E1 -27537.386,E2 -27537.386} C_VEL
LIN {X 0,Y 118.32,Z 443.668,A -85,B 0,C 180,E1 -27541.699,E2 -27541.699} C_VEL
LIN {X 0,Y 117.496,Z 444.765,A -85,B 0,C 180,E1 -27543.426,E2 -27543.426} C_VEL
LIN {X 0,Y 116.12,Z 445.97,A -85,B 0,C 180,E1 -27544.905,E2 -27544.905} C_VEL
LIN {X 0,Y 109.517,Z 449.673,A -85,B 0,C 180,E1 -27548.674,E2 -27548.674} C_VEL
LIN {X 0,Y 105.252,Z 451.686,A -85,B 0,C 180,E1 -27551.552,E2 -27551.552} C_VEL
LIN {X 0,Y 99.245,Z 453.736,A -85,B 0,C 180,E1 -27556.45,E2 -27556.45} C_VEL
LIN {X 0,Y 94.045,Z 454.711,A -85,B 0,C 180,E1 -27561.936,E2 -27561.936} C_VEL
LIN {X 0,Y 88.932,Z 454.486,A -85,B 0,C 180,E1 -27569.613,E2 -27569.613} C_VEL
LIN {X 0,Y 86.308,Z 453.335,A -85,B 0,C 180,E1 -27575.472,E2 -27575.472} C_VEL
LIN {X 0,Y 84.585,Z 451.328,A -85,B 0,C 180,E1 -27581.653,E2 -27581.653} C_VEL
LIN {X 0,Y 83.734,Z 447.893,A -85,B 0,C 180,E1 -27589.052,E2 -27589.052} C_VEL
LIN {X 0,Y 84.123,Z 442.835,A -85,B 0,C 180,E1 -27596.653,E2 -27596.653} C_VEL
LIN {X 0,Y 85.234,Z 437.811,A -85,B 0,C 180,E1 -27602.431,E2 -27602.431} C_VEL
LIN {X 0,Y 86.723,Z 432.437,A -85,B 0,C 180,E1 -27607.354,E2 -27607.354} C_VEL
LIN {X 0,Y 88.613,Z 425.939,A -85,B 0,C 180,E1 -27612.109,E2 -27612.109} C_VEL
LIN {X 0,Y 88.756,Z 425.518,A -85,B 0,C 180,E1 -27612.38,E2 -27612.38} C_VEL
LIN {X 0,Y 89.041,Z 422.354,A -85,B 0,C 180,E1 -27614.469,E2 -27614.469} C_VEL
LIN {X 0,Y 87.902,Z 418.133,A -85,B 0,C 180,E1 -27617.124,E2 -27617.124} C_VEL
LIN {X 0,Y 85.915,Z 412.267,A -85,B 0,C 180,E1 -27620.699,E2 -27620.699} C_VEL
LIN {X 0,Y 85.645,Z 410.131,A -85,B 0,C 180,E1 -27621.851,E2 -27621.851} C_VEL
LIN {X 0,Y 85.048,Z 399.979,A -85,B 0,C 180,E1 -27626.471,E2 -27626.471} C_VEL
LIN {X 0,Y 83.26,Z 391.737,A -85,B 0,C 180,E1 -27629.994,E2 -27629.994} C_VEL
LIN {X 0,Y 81.959,Z 387.3,A -85,B 0,C 180,E1 -27631.836,E2 -27631.836} C_VEL
LIN {X 0,Y 80.363,Z 383.929,A -85,B 0,C 180,E1 -27633.44,E2 -27633.44} C_VEL
LIN {X 0,Y 80.22,Z 383.306,A -85,B 0,C 180,E1 -27633.761,E2 -27633.761} C_VEL
LIN {X 0,Y 79.992,Z 383.329,A -85,B 0,C 180,E1 -27640.114,E2 -27640.114} C_VEL
LIN {X 0,Y 79.753,Z 383.363,A -85,B 0,C 180,E1 -27645.322,E2 -27645.322} C_VEL
LIN {X 0,Y 79.505,Z 383.387,A -85,B 0,C 180,E1 -27650.7,E2 -27650.7} C_VEL
LIN {X 0,Y 79.474,Z 383.39,A -85,B 0,C 180,E1 -27657.844,E2 -27657.844} C_VEL
LIN {X 0,Y 79.451,Z 383.393,A -85,B 0,C 180,E1 -27667.249,E2 -27667.249} C_VEL
LIN {X 0,Y 79.483,Z 383.389,A -85,B 0,C 180,E1 -27675.012,E2 -27675.012} C_VEL
LIN {X 0,Y 79.451,Z 383.393,A -85,B 0,C 180,E1 -27682.749,E2 -27682.749} C_VEL
LIN {X 0,Y 79.473,Z 383.391,A -85,B 0,C 180,E1 -27692.153,E2 -27692.153} C_VEL
LIN {X 0,Y 79.52,Z 383.384,A -85,B 0,C 180,E1 -27699.303,E2 -27699.303} C_VEL
LIN {X 0,Y 79.869,Z 383.347,A -85,B 0,C 180,E1 -27705.424,E2 -27705.424} C_VEL
LIN {X 0,Y 79.994,Z 383.33,A -85,B 0,C 180,E1 -27709.885,E2 -27709.885} C_VEL
LIN {X 0,Y 80.643,Z 383.253,A -85,B 0,C 180,E1 -27720.005,E2 -27720.005} C_VEL
LIN {X 0,Y 79.991,Z 383.332,A -85,B 0,C 180,E1 -27730.126,E2 -27730.126} C_VEL
LIN {X 0,Y 79.755,Z 383.361,A -85,B 0,C 180,E1 -27735.334,E2 -27735.334} C_VEL
LIN {X 0,Y 79.508,Z 383.386,A -85,B 0,C 180,E1 -27740.711,E2 -27740.711} C_VEL
LIN {X 0,Y 79.476,Z 383.393,A -85,B 0,C 180,E1 -27747.851,E2 -27747.851} C_VEL
LIN {X 0,Y 79.448,Z 383.393,A -85,B 0,C 180,E1 -27757.248,E2 -27757.248} C_VEL
LIN {X 0,Y 79.749,Z 383.52,A -85,B 0,C 180,E1 -27764.614,E2 -27764.614} C_VEL
LIN {X 0,Y 80.955,Z 386.411,A -85,B 0,C 180,E1 -27765.793,E2 -27765.793} C_VEL
LIN {X 0,Y 82.245,Z 389.222,A -85,B 0,C 180,E1 -27766.952,E2 -27766.952} C_VEL
LIN {X 0,Y 83.505,Z 394.379,A -85,B 0,C 180,E1 -27768.743,E2 -27768.743} C_VEL
LIN {X 0,Y 83.547,Z 403.577,A -85,B 0,C 180,E1 -27771.709,E2 -27771.709} C_VEL
LIN {X 0,Y 83.3,Z 412.139,A -85,B 0,C 180,E1 -27775.047,E2 -27775.047} C_VEL
LIN {X 0,Y 82.863,Z 419.51,A -85,B 0,C 180,E1 -27778.464,E2 -27778.464} C_VEL
LIN {X 0,Y 82.265,Z 427.1,A -85,B 0,C 180,E1 -27782.672,E2 -27782.672} C_VEL
LIN {X 0,Y 82.02,Z 430.3,A -85,B 0,C 180,E1 -27784.639,E2 -27784.639} C_VEL
LIN {X 0,Y 79.734,Z 438.417,A -85,B 0,C 180,E1 -27790.706,E2 -27790.706} C_VEL
LIN {X 0,Y 78.453,Z 443.709,A -85,B 0,C 180,E1 -27795.745,E2 -27795.745} C_VEL
LIN {X 0,Y 77.544,Z 449.041,A -85,B 0,C 180,E1 -27802.193,E2 -27802.193} C_VEL
LIN {X 0,Y 77.492,Z 452.521,A -85,B 0,C 180,E1 -27807.405,E2 -27807.405} C_VEL
LIN {X 0,Y 77.571,Z 453.97,A -85,B 0,C 180,E1 -27810.007,E2 -27810.007} C_VEL
LIN {X 0,Y 77.375,Z 456.334,A -85,B 0,C 180,E1 -27815.218,E2 -27815.218} C_VEL
LIN {X 0,Y 77.601,Z 458.191,A -85,B 0,C 180,E1 -27820.442,E2 -27820.442} C_VEL
LIN {X 0,Y 78.458,Z 459.57,A -85,B 0,C 180,E1 -27825.595,E2 -27825.595} C_VEL
LIN {X 0,Y 79.945,Z 460.38,A -85,B 0,C 180,E1 -27830.595,E2 -27830.595} C_VEL
LIN {X 0,Y 84.664,Z 460.807,A -85,B 0,C 180,E1 -27839.879,E2 -27839.879} C_VEL
LIN {X 0,Y 87.954,Z 460.369,A -85,B 0,C 180,E1 -27844.017,E2 -27844.017} C_VEL
LIN {X 0,Y 91.733,Z 459.402,A -85,B 0,C 180,E1 -27847.807,E2 -27847.807} C_VEL
LIN {X 0,Y 95.859,Z 458.023,A -85,B 0,C 180,E1 -27851.295,E2 -27851.295} C_VEL
LIN {X 0,Y 102.646,Z 455.08,A -85,B 0,C 180,E1 -27855.972,E2 -27855.972} C_VEL
LIN {X 0,Y 105.97,Z 453.201,A -85,B 0,C 180,E1 -27858.451,E2 -27858.451} C_VEL
LIN {X 0,Y 110.771,Z 449.709,A -85,B 0,C 180,E1 -27862.481,E2 -27862.481} C_VEL
LIN {X 0,Y 112,Z 447.754,A -85,B 0,C 180,E1 -27865.611,E2 -27865.611} C_VEL
LIN {X 0,Y 112.624,Z 446.558,A -85,B 0,C 180,E1 -27867.962,E2 -27867.962} C_VEL
LIN {X 0,Y 112.991,Z 445.506,A -85,B 0,C 180,E1 -27870.559,E2 -27870.559} C_VEL
LIN {X 0,Y 113.479,Z 444.194,A -85,B 0,C 180,E1 -27874.305,E2 -27874.305} C_VEL
LIN {X 0,Y 113.812,Z 443.206,A -85,B 0,C 180,E1 -27878.25,E2 -27878.25} C_VEL
LIN {X 0,Y 114.056,Z 442.643,A -85,B 0,C 180,E1 -27882.052,E2 -27882.052} C_VEL
LIN {X 0,Y 114.284,Z 442.51,A -85,B 0,C 180,E1 -27885.757,E2 -27885.757} C_VEL
LIN {X 0,Y 114.493,Z 442.68,A -85,B 0,C 180,E1 -27889.385,E2 -27889.385} C_VEL
LIN {X 0,Y 114.193,Z 443.4,A -85,B 0,C 180,E1 -27892.926,E2 -27892.926} C_VEL
LIN {X 0,Y 113.483,Z 444.527,A -85,B 0,C 180,E1 -27896.446,E2 -27896.446} C_VEL
LIN {X 0,Y 112.389,Z 446.096,A -85,B 0,C 180,E1 -27899.996,E2 -27899.996} C_VEL
LIN {X 0,Y 111.476,Z 446.957,A -85,B 0,C 180,E1 -27901.803,E2 -27901.803} C_VEL
LIN {X 0,Y 108.691,Z 448.623,A -85,B 0,C 180,E1 -27903.704,E2 -27903.704} C_VEL
LIN {X 0,Y 99.667,Z 452.548,A -85,B 0,C 180,E1 -27909.145,E2 -27909.145} C_VEL
LIN {X 0,Y 93.999,Z 454.224,A -85,B 0,C 180,E1 -27913.576,E2 -27913.576} C_VEL
LIN {X 0,Y 88.96,Z 455.074,A -85,B 0,C 180,E1 -27918.537,E2 -27918.537} C_VEL
LIN {X 0,Y 84.294,Z 455.043,A -85,B 0,C 180,E1 -27924.632,E2 -27924.632} C_VEL
LIN {X 0,Y 80.489,Z 453.969,A -85,B 0,C 180,E1 -27931.588,E2 -27931.588} C_VEL
LIN {X 0,Y 77.958,Z 451.817,A -85,B 0,C 180,E1 -27939.121,E2 -27939.121} C_VEL
LIN {X 0,Y 76.723,Z 448.482,A -85,B 0,C 180,E1 -27947.115,E2 -27947.115} C_VEL
LIN {X 0,Y 76.868,Z 443.597,A -85,B 0,C 180,E1 -27955.362,E2 -27955.362} C_VEL
LIN {X 0,Y 77.883,Z 438.647,A -85,B 0,C 180,E1 -27961.715,E2 -27961.715} C_VEL
LIN {X 0,Y 79.181,Z 434.107,A -85,B 0,C 180,E1 -27966.452,E2 -27966.452} C_VEL
LIN {X 0,Y 81.222,Z 427.219,A -85,B 0,C 180,E1 -27972.122,E2 -27972.122} C_VEL
LIN {X 0,Y 83.404,Z 420.318,A -85,B 0,C 180,E1 -27976.596,E2 -27976.596} C_VEL
LIN {X 0,Y 85.66,Z 412.635,A -85,B 0,C 180,E1 -27980.55,E2 -27980.55} C_VEL
LIN {X 0,Y 85.645,Z 410.131,A -85,B 0,C 180,E1 -27981.851,E2 -27981.851} C_VEL
LIN {X 0,Y 84.834,Z 405.484,A -85,B 0,C 180,E1 -27984.286,E2 -27984.286} C_VEL
LIN {X 0,Y 82.324,Z 399.551,A -85,B 0,C 180,E1 -27987.5,E2 -27987.5} C_VEL
LIN {X 0,Y 77.955,Z 392.501,A -85,B 0,C 180,E1 -27991.697,E2 -27991.697} C_VEL
LIN {X 0,Y 74.074,Z 386.993,A -85,B 0,C 180,E1 -27995.189,E2 -27995.189} C_VEL
LIN {X 0,Y 72.997,Z 384.205,A -85,B 0,C 180,E1 -27996.731,E2 -27996.731} C_VEL
LIN {X 0,Y 72.876,Z 384.212,A -85,B 0,C 180,E1 -28001.113,E2 -28001.113} C_VEL
LIN {X 0,Y 72.573,Z 384.257,A -85,B 0,C 180,E1 -28006.882,E2 -28006.882} C_VEL
LIN {X 0,Y 72.385,Z 384.28,A -85,B 0,C 180,E1 -28012.845,E2 -28012.845} C_VEL
LIN {X 0,Y 72.366,Z 384.276,A -85,B 0,C 180,E1 -28019.079,E2 -28019.079} C_VEL
LIN {X 0,Y 72.335,Z 384.28,A -85,B 0,C 180,E1 -28025.65,E2 -28025.65} C_VEL
LIN {X 0,Y 72.319,Z 384.285,A -85,B 0,C 180,E1 -28032.854,E2 -28032.854} C_VEL
LIN {X 0,Y 72.357,Z 384.281,A -85,B 0,C 180,E1 -28040.977,E2 -28040.977} C_VEL
LIN {X 0,Y 72.334,Z 384.282,A -85,B 0,C 180,E1 -28044.348,E2 -28044.348} C_VEL
LIN {X 0,Y 72.381,Z 384.273,A -85,B 0,C 180,E1 -28050.962,E2 -28050.962} C_VEL
LIN {X 0,Y 72.393,Z 384.278,A -85,B 0,C 180,E1 -28057.156,E2 -28057.156} C_VEL
LIN {X 0,Y 72.773,Z 384.231,A -85,B 0,C 180,E1 -28064.931,E2 -28064.931} C_VEL
LIN {X 0,Y 72.887,Z 384.212,A -85,B 0,C 180,E1 -28068.887,E2 -28068.887} C_VEL
LIN {X 0,Y 73.57,Z 384.134,A -85,B 0,C 180,E1 -28080.005,E2 -28080.005} C_VEL
LIN {X 0,Y 72.876,Z 384.214,A -85,B 0,C 180,E1 -28091.126,E2 -28091.126} C_VEL
LIN {X 0,Y 72.576,Z 384.257,A -85,B 0,C 180,E1 -28096.894,E2 -28096.894} C_VEL
LIN {X 0,Y 72.388,Z 384.277,A -85,B 0,C 180,E1 -28102.858,E2 -28102.858} C_VEL
LIN {X 0,Y 72.372,Z 384.275,A -85,B 0,C 180,E1 -28109.09,E2 -28109.09} C_VEL
LIN {X 0,Y 72.409,Z 384.273,A -85,B 0,C 180,E1 -28119.073,E2 -28119.073} C_VEL
LIN {X 0,Y 72.547,Z 384.461,A -85,B 0,C 180,E1 -28121.634,E2 -28121.634} C_VEL
LIN {X 0,Y 73.749,Z 387.327,A -85,B 0,C 180,E1 -28122.991,E2 -28122.991} C_VEL
LIN {X 0,Y 75.845,Z 391.224,A -85,B 0,C 180,E1 -28124.93,E2 -28124.93} C_VEL
LIN {X 0,Y 77.029,Z 395.796,A -85,B 0,C 180,E1 -28126.886,E2 -28126.886} C_VEL
LIN {X 0,Y 76.904,Z 404.995,A -85,B 0,C 180,E1 -28130.239,E2 -28130.239} C_VEL
LIN {X 0,Y 76.462,Z 413.85,A -85,B 0,C 180,E1 -28134.141,E2 -28134.141} C_VEL
LIN {X 0,Y 75.691,Z 423.432,A -85,B 0,C 180,E1 -28139.299,E2 -28139.299} C_VEL
LIN {X 0,Y 75.028,Z 429.906,A -85,B 0,C 180,E1 -28143.588,E2 -28143.588} C_VEL
LIN {X 0,Y 72.676,Z 438.05,A -85,B 0,C 180,E1 -28150.225,E2 -28150.225} C_VEL
LIN {X 0,Y 71.357,Z 443.344,A -85,B 0,C 180,E1 -28155.753,E2 -28155.753} C_VEL
LIN {X 0,Y 70.569,Z 447.747,A -85,B 0,C 180,E1 -28161.416,E2 -28161.416} C_VEL
LIN {X 0,Y 70.467,Z 451.913,A -85,B 0,C 180,E1 -28168.111,E2 -28168.111} C_VEL
LIN {X 0,Y 70.43,Z 454.629,A -85,B 0,C 180,E1 -28173.659,E2 -28173.659} C_VEL
LIN {X 0,Y 70.66,Z 457.4,A -85,B 0,C 180,E1 -28181.482,E2 -28181.482} C_VEL
LIN {X 0,Y 71.665,Z 458.806,A -85,B 0,C 180,E1 -28187.117,E2 -28187.117} C_VEL
LIN {X 0,Y 75.667,Z 460.359,A -85,B 0,C 180,E1 -28197.679,E2 -28197.679} C_VEL
LIN {X 0,Y 78.581,Z 460.51,A -85,B 0,C 180,E1 -28202.461,E2 -28202.461} C_VEL
LIN {X 0,Y 82.162,Z 460.123,A -85,B 0,C 180,E1 -28206.789,E2 -28206.789} C_VEL
LIN {X 0,Y 90.641,Z 458.161,A -85,B 0,C 180,E1 -28214.261,E2 -28214.261} C_VEL
LIN {X 0,Y 97.804,Z 455.423,A -85,B 0,C 180,E1 -28218.99,E2 -28218.99} C_VEL
LIN {X 0,Y 102.203,Z 453.135,A -85,B 0,C 180,E1 -28222.264,E2 -28222.264} C_VEL
LIN {X 0,Y 104.315,Z 451.729,A -85,B 0,C 180,E1 -28223.955,E2 -28223.955} C_VEL
LIN {X 0,Y 106.066,Z 449.788,A -85,B 0,C 180,E1 -28227.985,E2 -28227.985} C_VEL
LIN {X 0,Y 106.887,Z 448.149,A -85,B 0,C 180,E1 -28232.592,E2 -28232.592} C_VEL
LIN {X 0,Y 107.42,Z 447.006,A -85,B 0,C 180,E1 -28236.883,E2 -28236.883} C_VEL
LIN {X 0,Y 107.747,Z 446.32,A -85,B 0,C 180,E1 -28240.962,E2 -28240.962} C_VEL
LIN {X 0,Y 108.138,Z 446.029,A -85,B 0,C 180,E1 -28247.146,E2 -28247.146} C_VEL
LIN {X 0,Y 108.223,Z 446.079,A -85,B 0,C 180,E1 -28248.762,E2 -28248.762} C_VEL
LIN {X 0,Y 107.949,Z 446.676,A -85,B 0,C 180,E1 -28252.515,E2 -28252.515} C_VEL
LIN {X 0,Y 106.978,Z 447.648,A -85,B 0,C 180,E1 -28256.23,E2 -28256.23} C_VEL
LIN {X 0,Y 105.348,Z 449.052,A -85,B 0,C 180,E1 -28259.996,E2 -28259.996} C_VEL
LIN {X 0,Y 98.615,Z 452.002,A -85,B 0,C 180,E1 -28263.787,E2 -28263.787} C_VEL
LIN {X 0,Y 90.908,Z 454.384,A -85,B 0,C 180,E1 -28268.89,E2 -28268.89} C_VEL
LIN {X 0,Y 84.468,Z 455.429,A -85,B 0,C 180,E1 -28274.449,E2 -28274.449} C_VEL
LIN {X 0,Y 79.05,Z 455.435,A -85,B 0,C 180,E1 -28280.826,E2 -28280.826} C_VEL
LIN {X 0,Y 74.627,Z 454.4,A -85,B 0,C 180,E1 -28288.085,E2 -28288.085} C_VEL
LIN {X 0,Y 71.102,Z 451.801,A -85,B 0,C 180,E1 -28297.733,E2 -28297.733} C_VEL
LIN {X 0,Y 69.791,Z 448.855,A -85,B 0,C 180,E1 -28305.168,E2 -28305.168} C_VEL
LIN {X 0,Y 69.662,Z 444.307,A -85,B 0,C 180,E1 -28313.802,E2 -28313.802} C_VEL
LIN {X 0,Y 70.719,Z 438.724,A -85,B 0,C 180,E1 -28321.732,E2 -28321.732} C_VEL
LIN {X 0,Y 72.546,Z 432.587,A -85,B 0,C 180,E1 -28328.453,E2 -28328.453} C_VEL
LIN {X 0,Y 74.413,Z 426.691,A -85,B 0,C 180,E1 -28333.534,E2 -28333.534} C_VEL
LIN {X 0,Y 76.63,Z 420.071,A -85,B 0,C 180,E1 -28338.084,E2 -28338.084} C_VEL
LIN {X 0,Y 78.826,Z 413.175,A -85,B 0,C 180,E1 -28341.878,E2 -28341.878} C_VEL
LIN {X 0,Y 78.671,Z 406.193,A -85,B 0,C 180,E1 -28345.623,E2 -28345.623} C_VEL
LIN {X 0,Y 78.227,Z 400.382,A -85,B 0,C 180,E1 -28348.49,E2 -28348.49} C_VEL
LIN {X 0,Y 76.319,Z 391.606,A -85,B 0,C 180,E1 -28352.63,E2 -28352.63} C_VEL
LIN {X 0,Y 74.074,Z 386.993,A -85,B 0,C 180,E1 -28355.189,E2 -28355.189} C_VEL
LIN {X 0,Y 72.253,Z 385.194,A -85,B 0,C 180,E1 -28357.265,E2 -28357.265} C_VEL
LIN {X 0,Y 70.218,Z 384.545,A -85,B 0,C 180,E1 -28360.214,E2 -28360.214} C_VEL
LIN {X 0,Y 66.362,Z 385.123,A -85,B 0,C 180,E1 -28369.434,E2 -28369.434} C_VEL
LIN {X 0,Y 65.249,Z 385.167,A -85,B 0,C 180,E1 -28380.477,E2 -28380.477} C_VEL
LIN {X 0,Y 65.253,Z 385.169,A -85,B 0,C 180,E1 -28391.079,E2 -28391.079} C_VEL
LIN {X 0,Y 65.269,Z 385.167,A -85,B 0,C 180,E1 -28399.763,E2 -28399.763} C_VEL
LIN {X 0,Y 65.25,Z 385.165,A -85,B 0,C 180,E1 -28409.489,E2 -28409.489} C_VEL
LIN {X 0,Y 65.241,Z 385.17,A -85,B 0,C 180,E1 -28414.483,E2 -28414.483} C_VEL
LIN {X 0,Y 65.661,Z 385.118,A -85,B 0,C 180,E1 -28424.4,E2 -28424.4} C_VEL
LIN {X 0,Y 65.789,Z 385.094,A -85,B 0,C 180,E1 -28427.67,E2 -28427.67} C_VEL
LIN {X 0,Y 66.494,Z 385.015,A -85,B 0,C 180,E1 -28440.006,E2 -28440.006} C_VEL
LIN {X 0,Y 65.767,Z 385.096,A -85,B 0,C 180,E1 -28452.347,E2 -28452.347} C_VEL
LIN {X 0,Y 65.379,Z 385.15,A -85,B 0,C 180,E1 -28458.82,E2 -28458.82} C_VEL
LIN {X 0,Y 65.234,Z 385.172,A -85,B 0,C 180,E1 -28465.534,E2 -28465.534} C_VEL
LIN {X 0,Y 65.21,Z 385.174,A -85,B 0,C 180,E1 -28472.614,E2 -28472.614} C_VEL
LIN {X 0,Y 65.318,Z 385.205,A -85,B 0,C 180,E1 -28477.86,E2 -28477.86} C_VEL
LIN {X 0,Y 66.412,Z 388.034,A -85,B 0,C 180,E1 -28479.423,E2 -28479.423} C_VEL
LIN {X 0,Y 69.985,Z 394.939,A -85,B 0,C 180,E1 -28483.655,E2 -28483.655} C_VEL
LIN {X 0,Y 70.657,Z 398.693,A -85,B 0,C 180,E1 -28485.336,E2 -28485.336} C_VEL
LIN {X 0,Y 70.016,Z 410.01,A -85,B 0,C 180,E1 -28490.225,E2 -28490.225} C_VEL
LIN {X 0,Y 69.319,Z 418.369,A -85,B 0,C 180,E1 -28494.757,E2 -28494.757} C_VEL
LIN {X 0,Y 68.465,Z 426.311,A -85,B 0,C 180,E1 -28499.981,E2 -28499.981} C_VEL
LIN {X 0,Y 67.645,Z 431.318,A -85,B 0,C 180,E1 -28503.805,E2 -28503.805} C_VEL
LIN {X 0,Y 65.63,Z 437.659,A -85,B 0,C 180,E1 -28509.642,E2 -28509.642} C_VEL
